	VAR robtarget OpenholeUD_3424 := [[417.35, -17.1, 182.09], [-0.110581, 0.698407, 0.70005, 0.099652], [0,0,0,0], [9E9, 9E9, 9E9, 9E9, 9E9, 9E9]];
	VAR robtarget OpenholeUD_3425 := [[421.34, -17.1, 182.02], [-0.098166, 0.70026, 0.701711, 0.087187], [0,0,0,0], [9E9, 9E9, 9E9, 9E9, 9E9, 9E9]];
	VAR robtarget OpenholeUD_3426 := [[425.34, -17.1, 181.95], [-0.085471, 0.701922, 0.703176, 0.074457], [0,0,0,0], [9E9, 9E9, 9E9, 9E9, 9E9, 9E9]];
	VAR robtarget OpenholeUD_3427 := [[429.34, -17.1, 181.87], [-0.072525, 0.703378, 0.704428, 0.061492], [0,0,0,0], [9E9, 9E9, 9E9, 9E9, 9E9, 9E9]];
	VAR robtarget OpenholeUD_3428 := [[433.34, -17.1, 181.8], [-0.059361, 0.704611, 0.705453, 0.048326], [0,0,0,0], [9E9, 9E9, 9E9, 9E9, 9E9, 9E9]];
	VAR robtarget OpenholeUD_3429 := [[437.34, -17.1, 181.72], [-0.046017, 0.705608, 0.70624, 0.034996], [0,0,0,0], [9E9, 9E9, 9E9, 9E9, 9E9, 9E9]];
	VAR robtarget OpenholeUD_3430 := [[443.05, -17.1, 181.62], [-0.02675, 0.706601, 0.706931, 0.015776], [0,0,0,0], [9E9, 9E9, 9E9, 9E9, 9E9, 9E9]];
	VAR robtarget OpenholeUD_3431 := [[443.05, -17.1, 181.62], [-0.02675, 0.706601, 0.706931, 0.015776], [0,0,0,0], [9E9, 9E9, 9E9, 9E9, 9E9, 9E9]];
	VAR robtarget OpenholeUD_3432 := [[443.48, -15.9, 181.68], [-0.029359, 0.706497, 0.707033, 0.010242], [0,0,0,0], [9E9, 9E9, 9E9, 9E9, 9E9, 9E9]];
	VAR robtarget OpenholeUD_3433 := [[439.48, -15.9, 181.8], [-0.042881, 0.705805, 0.706708, 0.023756], [0,0,0,0], [9E9, 9E9, 9E9, 9E9, 9E9, 9E9]];
	VAR robtarget OpenholeUD_3434 := [[435.48, -15.9, 181.92], [-0.056278, 0.704864, 0.706129, 0.037174], [0,0,0,0], [9E9, 9E9, 9E9, 9E9, 9E9, 9E9]];
	VAR robtarget OpenholeUD_3435 := [[431.49, -15.9, 182.04], [-0.06951, 0.703682, 0.705304, 0.050457], [0,0,0,0], [9E9, 9E9, 9E9, 9E9, 9E9, 9E9]];
	VAR robtarget OpenholeUD_3436 := [[427.49, -15.9, 182.16], [-0.082538, 0.702273, 0.704244, 0.063565], [0,0,0,0], [9E9, 9E9, 9E9, 9E9, 9E9, 9E9]];
	VAR robtarget OpenholeUD_3437 := [[423.49, -15.9, 182.28], [-0.095326, 0.700652, 0.702961, 0.076462], [0,0,0,0], [9E9, 9E9, 9E9, 9E9, 9E9, 9E9]];
	VAR robtarget OpenholeUD_3438 := [[419.49, -15.9, 182.4], [-0.107844, 0.698835, 0.701469, 0.089115], [0,0,0,0], [9E9, 9E9, 9E9, 9E9, 9E9, 9E9]];
	VAR robtarget OpenholeUD_3439 := [[415.49, -15.9, 182.52], [-0.120064, 0.696839, 0.699785, 0.101497], [0,0,0,0], [9E9, 9E9, 9E9, 9E9, 9E9, 9E9]];
	VAR robtarget OpenholeUD_3440 := [[411.5, -15.9, 182.64], [-0.131964, 0.694684, 0.697925, 0.113581], [0,0,0,0], [9E9, 9E9, 9E9, 9E9, 9E9, 9E9]];
	VAR robtarget OpenholeUD_3441 := [[407.5, -15.9, 182.76], [-0.143525, 0.692388, 0.695908, 0.125349], [0,0,0,0], [9E9, 9E9, 9E9, 9E9, 9E9, 9E9]];
	VAR robtarget OpenholeUD_3442 := [[403.5, -15.9, 182.88], [-0.154733, 0.689969, 0.693751, 0.136783], [0,0,0,0], [9E9, 9E9, 9E9, 9E9, 9E9, 9E9]];
	VAR robtarget OpenholeUD_3443 := [[399.5, -15.9, 183], [-0.165579, 0.687447, 0.691472, 0.147872], [0,0,0,0], [9E9, 9E9, 9E9, 9E9, 9E9, 9E9]];
	VAR robtarget OpenholeUD_3444 := [[395.5, -15.9, 183.12], [-0.176055, 0.684839, 0.689089, 0.158607], [0,0,0,0], [9E9, 9E9, 9E9, 9E9, 9E9, 9E9]];
	VAR robtarget OpenholeUD_3445 := [[389.35, -15.9, 183.31], [-0.191445, 0.680697, 0.685258, 0.174418], [0,0,0,0], [9E9, 9E9, 9E9, 9E9, 9E9, 9E9]];
	VAR robtarget OpenholeUD_3446 := [[385.35, -15.9, 183.32], [-0.183051, 0.683002, 0.683002, 0.183051], [0,0,0,0], [9E9, 9E9, 9E9, 9E9, 9E9, 9E9]];
	VAR robtarget OpenholeUD_3447 := [[381.35, -15.9, 183.33], [-0.183051, 0.683002, 0.683002, 0.183051], [0,0,0,0], [9E9, 9E9, 9E9, 9E9, 9E9, 9E9]];
	VAR robtarget OpenholeUD_3448 := [[377.35, -15.9, 183.34], [-0.183051, 0.683002, 0.683002, 0.183051], [0,0,0,0], [9E9, 9E9, 9E9, 9E9, 9E9, 9E9]];
	VAR robtarget OpenholeUD_3449 := [[369.35, -15.9, 183.37], [-0.183051, 0.683002, 0.683002, 0.183051], [0,0,0,0], [9E9, 9E9, 9E9, 9E9, 9E9, 9E9]];
	VAR robtarget OpenholeUD_3450 := [[369.35, -15.9, 183.37], [-0.183051, 0.683002, 0.683002, 0.183051], [0,0,0,0], [9E9, 9E9, 9E9, 9E9, 9E9, 9E9]];
	VAR robtarget OpenholeUD_3451 := [[369.35, -14.7, 184.06], [-0.183051, 0.683002, 0.683002, 0.183051], [0,0,0,0], [9E9, 9E9, 9E9, 9E9, 9E9, 9E9]];
	VAR robtarget OpenholeUD_3452 := [[373.35, -14.7, 184.05], [-0.183051, 0.683002, 0.683002, 0.183051], [0,0,0,0], [9E9, 9E9, 9E9, 9E9, 9E9, 9E9]];
	VAR robtarget OpenholeUD_3453 := [[377.35, -14.7, 184.04], [-0.183051, 0.683002, 0.683002, 0.183051], [0,0,0,0], [9E9, 9E9, 9E9, 9E9, 9E9, 9E9]];
	VAR robtarget OpenholeUD_3454 := [[381.35, -14.7, 184.03], [-0.183051, 0.683002, 0.683002, 0.183051], [0,0,0,0], [9E9, 9E9, 9E9, 9E9, 9E9, 9E9]];
	VAR robtarget OpenholeUD_3455 := [[389.35, -14.7, 184], [-0.194849, 0.679731, 0.68612, 0.170995], [0,0,0,0], [9E9, 9E9, 9E9, 9E9, 9E9, 9E9]];
	VAR robtarget OpenholeUD_3456 := [[393.35, -14.7, 183.83], [-0.185019, 0.682472, 0.688592, 0.16075], [0,0,0,0], [9E9, 9E9, 9E9, 9E9, 9E9, 9E9]];
	VAR robtarget OpenholeUD_3457 := [[397.35, -14.7, 183.67], [-0.174817, 0.685156, 0.690982, 0.150146], [0,0,0,0], [9E9, 9E9, 9E9, 9E9, 9E9, 9E9]];
	VAR robtarget OpenholeUD_3458 := [[401.34, -14.7, 183.5], [-0.164241, 0.687768, 0.693273, 0.139186], [0,0,0,0], [9E9, 9E9, 9E9, 9E9, 9E9, 9E9]];
	VAR robtarget OpenholeUD_3459 := [[405.34, -14.7, 183.33], [-0.153297, 0.69029, 0.695448, 0.127878], [0,0,0,0], [9E9, 9E9, 9E9, 9E9, 9E9, 9E9]];
	VAR robtarget OpenholeUD_3460 := [[409.34, -14.7, 183.17], [-0.141992, 0.692704, 0.697488, 0.116232], [0,0,0,0], [9E9, 9E9, 9E9, 9E9, 9E9, 9E9]];
	VAR robtarget OpenholeUD_3461 := [[413.33, -14.7, 183], [-0.130337, 0.694991, 0.699378, 0.104265], [0,0,0,0], [9E9, 9E9, 9E9, 9E9, 9E9, 9E9]];
	VAR robtarget OpenholeUD_3462 := [[417.33, -14.7, 182.83], [-0.118347, 0.697133, 0.701097, 0.091993], [0,0,0,0], [9E9, 9E9, 9E9, 9E9, 9E9, 9E9]];
	VAR robtarget OpenholeUD_3463 := [[421.33, -14.7, 182.67], [-0.106043, 0.69911, 0.70263, 0.07944], [0,0,0,0], [9E9, 9E9, 9E9, 9E9, 9E9, 9E9]];
	VAR robtarget OpenholeUD_3464 := [[425.32, -14.7, 182.5], [-0.093448, 0.700905, 0.70396, 0.066634], [0,0,0,0], [9E9, 9E9, 9E9, 9E9, 9E9, 9E9]];
	VAR robtarget OpenholeUD_3465 := [[429.32, -14.7, 182.34], [-0.080591, 0.702499, 0.705072, 0.053604], [0,0,0,0], [9E9, 9E9, 9E9, 9E9, 9E9, 9E9]];
	VAR robtarget OpenholeUD_3466 := [[433.32, -14.7, 182.17], [-0.067504, 0.703877, 0.705953, 0.040385], [0,0,0,0], [9E9, 9E9, 9E9, 9E9, 9E9, 9E9]];
	VAR robtarget OpenholeUD_3467 := [[437.31, -14.7, 182], [-0.054224, 0.705025, 0.706591, 0.027016], [0,0,0,0], [9E9, 9E9, 9E9, 9E9, 9E9, 9E9]];
	VAR robtarget OpenholeUD_3468 := [[444.22, -14.7, 181.71], [-0.030919, 0.70643, 0.707097, 0.003662], [0,0,0,0], [9E9, 9E9, 9E9, 9E9, 9E9, 9E9]];
	VAR robtarget OpenholeUD_3469 := [[444.22, -14.7, 181.71], [-0.030919, 0.70643, 0.707097, 0.003662], [0,0,0,0], [9E9, 9E9, 9E9, 9E9, 9E9, 9E9]];
	VAR robtarget OpenholeUD_3470 := [[445.45, -13.5, 181.71], [-0.030843, 0.706434, 0.707092, -0.004551], [0,0,0,0], [9E9, 9E9, 9E9, 9E9, 9E9, 9E9]];
	VAR robtarget OpenholeUD_3471 := [[441.45, -13.5, 181.92], [-0.044373, 0.705713, 0.70705, 0.009], [0,0,0,0], [9E9, 9E9, 9E9, 9E9, 9E9, 9E9]];
	VAR robtarget OpenholeUD_3472 := [[437.46, -13.5, 182.13], [-0.057785, 0.704742, 0.706749, 0.022491], [0,0,0,0], [9E9, 9E9, 9E9, 9E9, 9E9, 9E9]];
	VAR robtarget OpenholeUD_3473 := [[433.46, -13.5, 182.35], [-0.071038, 0.703529, 0.706196, 0.035882], [0,0,0,0], [9E9, 9E9, 9E9, 9E9, 9E9, 9E9]];
	VAR robtarget OpenholeUD_3474 := [[429.47, -13.5, 182.56], [-0.084092, 0.702089, 0.705398, 0.04913], [0,0,0,0], [9E9, 9E9, 9E9, 9E9, 9E9, 9E9]];
	VAR robtarget OpenholeUD_3475 := [[425.48, -13.5, 182.77], [-0.096912, 0.700434, 0.704366, 0.062197], [0,0,0,0], [9E9, 9E9, 9E9, 9E9, 9E9, 9E9]];
	VAR robtarget OpenholeUD_3476 := [[421.48, -13.5, 182.98], [-0.109465, 0.698582, 0.703113, 0.075049], [0,0,0,0], [9E9, 9E9, 9E9, 9E9, 9E9, 9E9]];
	VAR robtarget OpenholeUD_3477 := [[417.49, -13.5, 183.2], [-0.121724, 0.696551, 0.701653, 0.087653], [0,0,0,0], [9E9, 9E9, 9E9, 9E9, 9E9, 9E9]];
	VAR robtarget OpenholeUD_3478 := [[413.49, -13.5, 183.41], [-0.133665, 0.694358, 0.700003, 0.099981], [0,0,0,0], [9E9, 9E9, 9E9, 9E9, 9E9, 9E9]];
	VAR robtarget OpenholeUD_3479 := [[409.5, -13.5, 183.62], [-0.145268, 0.692024, 0.698179, 0.112012], [0,0,0,0], [9E9, 9E9, 9E9, 9E9, 9E9, 9E9]];
	VAR robtarget OpenholeUD_3480 := [[405.5, -13.5, 183.83], [-0.156519, 0.689566, 0.696199, 0.123724], [0,0,0,0], [9E9, 9E9, 9E9, 9E9, 9E9, 9E9]];
	VAR robtarget OpenholeUD_3481 := [[401.51, -13.5, 184.05], [-0.167407, 0.687004, 0.69408, 0.135103], [0,0,0,0], [9E9, 9E9, 9E9, 9E9, 9E9, 9E9]];
	VAR robtarget OpenholeUD_3482 := [[397.51, -13.5, 184.26], [-0.177925, 0.684356, 0.691841, 0.146136], [0,0,0,0], [9E9, 9E9, 9E9, 9E9, 9E9, 9E9]];
	VAR robtarget OpenholeUD_3483 := [[393.52, -13.5, 184.47], [-0.188069, 0.681638, 0.689499, 0.156817], [0,0,0,0], [9E9, 9E9, 9E9, 9E9, 9E9, 9E9]];
	VAR robtarget OpenholeUD_3484 := [[389.36, -13.5, 184.69], [-0.198245, 0.678748, 0.686964, 0.167571], [0,0,0,0], [9E9, 9E9, 9E9, 9E9, 9E9, 9E9]];
	VAR robtarget OpenholeUD_3485 := [[385.36, -13.5, 184.71], [-0.183051, 0.683002, 0.683002, 0.183051], [0,0,0,0], [9E9, 9E9, 9E9, 9E9, 9E9, 9E9]];
	VAR robtarget OpenholeUD_3486 := [[381.36, -13.5, 184.72], [-0.183051, 0.683002, 0.683002, 0.183051], [0,0,0,0], [9E9, 9E9, 9E9, 9E9, 9E9, 9E9]];
	VAR robtarget OpenholeUD_3487 := [[377.36, -13.5, 184.73], [-0.183051, 0.683002, 0.683002, 0.183051], [0,0,0,0], [9E9, 9E9, 9E9, 9E9, 9E9, 9E9]];
	VAR robtarget OpenholeUD_3488 := [[373.36, -13.5, 184.74], [-0.183051, 0.683002, 0.683002, 0.183051], [0,0,0,0], [9E9, 9E9, 9E9, 9E9, 9E9, 9E9]];
	VAR robtarget OpenholeUD_3489 := [[369.36, -13.5, 184.76], [-0.183051, 0.683002, 0.683002, 0.183051], [0,0,0,0], [9E9, 9E9, 9E9, 9E9, 9E9, 9E9]];
	VAR robtarget OpenholeUD_3490 := [[369.36, -13.5, 184.76], [-0.183051, 0.683002, 0.683002, 0.183051], [0,0,0,0], [9E9, 9E9, 9E9, 9E9, 9E9, 9E9]];
	VAR robtarget OpenholeUD_3491 := [[369.36, -12.3, 185.45], [-0.183051, 0.683002, 0.683002, 0.183051], [0,0,0,0], [9E9, 9E9, 9E9, 9E9, 9E9, 9E9]];
	VAR robtarget OpenholeUD_3492 := [[373.36, -12.3, 185.44], [-0.183051, 0.683002, 0.683002, 0.183051], [0,0,0,0], [9E9, 9E9, 9E9, 9E9, 9E9, 9E9]];
	VAR robtarget OpenholeUD_3493 := [[377.36, -12.3, 185.42], [-0.183051, 0.683002, 0.683002, 0.183051], [0,0,0,0], [9E9, 9E9, 9E9, 9E9, 9E9, 9E9]];
	VAR robtarget OpenholeUD_3494 := [[381.36, -12.3, 185.41], [-0.183051, 0.683002, 0.683002, 0.183051], [0,0,0,0], [9E9, 9E9, 9E9, 9E9, 9E9, 9E9]];
	VAR robtarget OpenholeUD_3495 := [[385.36, -12.3, 185.4], [-0.183051, 0.683002, 0.683002, 0.183051], [0,0,0,0], [9E9, 9E9, 9E9, 9E9, 9E9, 9E9]];
	VAR robtarget OpenholeUD_3496 := [[389.36, -12.3, 185.39], [-0.201634, 0.677749, 0.687791, 0.164145], [0,0,0,0], [9E9, 9E9, 9E9, 9E9, 9E9, 9E9]];
	VAR robtarget OpenholeUD_3497 := [[393.35, -12.3, 185.13], [-0.191956, 0.680553, 0.690183, 0.153776], [0,0,0,0], [9E9, 9E9, 9E9, 9E9, 9E9, 9E9]];
	VAR robtarget OpenholeUD_3498 := [[397.34, -12.3, 184.87], [-0.181904, 0.683309, 0.692486, 0.143051], [0,0,0,0], [9E9, 9E9, 9E9, 9E9, 9E9, 9E9]];
	VAR robtarget OpenholeUD_3499 := [[401.33, -12.3, 184.61], [-0.171477, 0.686, 0.694682, 0.131975], [0,0,0,0], [9E9, 9E9, 9E9, 9E9, 9E9, 9E9]];
	VAR robtarget OpenholeUD_3500 := [[405.33, -12.3, 184.35], [-0.160678, 0.688609, 0.696754, 0.120556], [0,0,0,0], [9E9, 9E9, 9E9, 9E9, 9E9, 9E9]];
	VAR robtarget OpenholeUD_3501 := [[409.32, -12.3, 184.09], [-0.149513, 0.691119, 0.698685, 0.108807], [0,0,0,0], [9E9, 9E9, 9E9, 9E9, 9E9, 9E9]];
	VAR robtarget OpenholeUD_3502 := [[413.31, -12.3, 183.84], [-0.137992, 0.693511, 0.700458, 0.096743], [0,0,0,0], [9E9, 9E9, 9E9, 9E9, 9E9, 9E9]];
	VAR robtarget OpenholeUD_3503 := [[417.3, -12.3, 183.58], [-0.12613, 0.695767, 0.702054, 0.084384], [0,0,0,0], [9E9, 9E9, 9E9, 9E9, 9E9, 9E9]];
	VAR robtarget OpenholeUD_3504 := [[421.29, -12.3, 183.32], [-0.113945, 0.697866, 0.703457, 0.071753], [0,0,0,0], [9E9, 9E9, 9E9, 9E9, 9E9, 9E9]];
	VAR robtarget OpenholeUD_3505 := [[425.28, -12.3, 183.06], [-0.10146, 0.69979, 0.704651, 0.058879], [0,0,0,0], [9E9, 9E9, 9E9, 9E9, 9E9, 9E9]];
	VAR robtarget OpenholeUD_3506 := [[429.28, -12.3, 182.8], [-0.088701, 0.701521, 0.705622, 0.045794], [0,0,0,0], [9E9, 9E9, 9E9, 9E9, 9E9, 9E9]];
	VAR robtarget OpenholeUD_3507 := [[433.27, -12.3, 182.54], [-0.0757, 0.703043, 0.706358, 0.032532], [0,0,0,0], [9E9, 9E9, 9E9, 9E9, 9E9, 9E9]];
	VAR robtarget OpenholeUD_3508 := [[437.26, -12.3, 182.28], [-0.062492, 0.70434, 0.706848, 0.019133], [0,0,0,0], [9E9, 9E9, 9E9, 9E9, 9E9, 9E9]];
	VAR robtarget OpenholeUD_3509 := [[441.25, -12.3, 182.03], [-0.049116, 0.705399, 0.707084, 0.005638], [0,0,0,0], [9E9, 9E9, 9E9, 9E9, 9E9, 9E9]];
	VAR robtarget OpenholeUD_3510 := [[445.24, -12.3, 181.77], [-0.035614, 0.706209, 0.707063, -0.007911], [0,0,0,0], [9E9, 9E9, 9E9, 9E9, 9E9, 9E9]];
	VAR robtarget OpenholeUD_3511 := [[449.23, -12.3, 181.51], [-0.022029, 0.706764, 0.706781, -0.021469], [0,0,0,0], [9E9, 9E9, 9E9, 9E9, 9E9, 9E9]];
	VAR robtarget OpenholeUD_3512 := [[453.22, -12.3, 181.25], [-0.008405, 0.707057, 0.706241, -0.034991], [0,0,0,0], [9E9, 9E9, 9E9, 9E9, 9E9, 9E9]];
	VAR robtarget OpenholeUD_3513 := [[457.22, -12.3, 180.99], [0.00521, 0.707088, 0.705446, -0.048433], [0,0,0,0], [9E9, 9E9, 9E9, 9E9, 9E9, 9E9]];
	VAR robtarget OpenholeUD_3514 := [[461.21, -12.3, 180.73], [0.018773, 0.706858, 0.704405, -0.061753], [0,0,0,0], [9E9, 9E9, 9E9, 9E9, 9E9, 9E9]];
	VAR robtarget OpenholeUD_3515 := [[465.2, -12.3, 180.47], [0.032238, 0.706372, 0.703128, -0.074909], [0,0,0,0], [9E9, 9E9, 9E9, 9E9, 9E9, 9E9]];
	VAR robtarget OpenholeUD_3516 := [[469.19, -12.3, 180.22], [0.045564, 0.705637, 0.701627, -0.087863], [0,0,0,0], [9E9, 9E9, 9E9, 9E9, 9E9, 9E9]];
	VAR robtarget OpenholeUD_3517 := [[473.18, -12.3, 179.96], [0.058713, 0.704665, 0.699917, -0.100581], [0,0,0,0], [9E9, 9E9, 9E9, 9E9, 9E9, 9E9]];
	VAR robtarget OpenholeUD_3518 := [[477.17, -12.3, 179.7], [0.071646, 0.703468, 0.698014, -0.113032], [0,0,0,0], [9E9, 9E9, 9E9, 9E9, 9E9, 9E9]];
	VAR robtarget OpenholeUD_3519 := [[481.17, -12.3, 179.44], [0.084333, 0.70206, 0.695937, -0.125188], [0,0,0,0], [9E9, 9E9, 9E9, 9E9, 9E9, 9E9]];
	VAR robtarget OpenholeUD_3520 := [[485.16, -12.3, 179.18], [0.096745, 0.700457, 0.693703, -0.137027], [0,0,0,0], [9E9, 9E9, 9E9, 9E9, 9E9, 9E9]];
	VAR robtarget OpenholeUD_3521 := [[489.15, -12.3, 178.92], [0.108857, 0.698677, 0.691331, -0.14853], [0,0,0,0], [9E9, 9E9, 9E9, 9E9, 9E9, 9E9]];
	VAR robtarget OpenholeUD_3522 := [[493.14, -12.3, 178.67], [0.12065, 0.696738, 0.68884, -0.159683], [0,0,0,0], [9E9, 9E9, 9E9, 9E9, 9E9, 9E9]];
	VAR robtarget OpenholeUD_3523 := [[497.13, -12.3, 178.41], [0.132108, 0.694656, 0.686249, -0.170476], [0,0,0,0], [9E9, 9E9, 9E9, 9E9, 9E9, 9E9]];
	VAR robtarget OpenholeUD_3524 := [[501.12, -12.3, 178.15], [0.143219, 0.692451, 0.683575, -0.180902], [0,0,0,0], [9E9, 9E9, 9E9, 9E9, 9E9, 9E9]];
	VAR robtarget OpenholeUD_3525 := [[505.12, -12.3, 177.89], [0.153974, 0.690139, 0.680835, -0.190956], [0,0,0,0], [9E9, 9E9, 9E9, 9E9, 9E9, 9E9]];
	VAR robtarget OpenholeUD_3526 := [[509.33, -12.3, 177.62], [0.183051, 0.683002, 0.683002, -0.183051], [0,0,0,0], [9E9, 9E9, 9E9, 9E9, 9E9, 9E9]];
	VAR robtarget OpenholeUD_3527 := [[513.33, -12.3, 177.6], [0.183051, 0.683002, 0.683002, -0.183051], [0,0,0,0], [9E9, 9E9, 9E9, 9E9, 9E9, 9E9]];
	VAR robtarget OpenholeUD_3528 := [[517.33, -12.3, 177.59], [0.183051, 0.683002, 0.683002, -0.183051], [0,0,0,0], [9E9, 9E9, 9E9, 9E9, 9E9, 9E9]];
	VAR robtarget OpenholeUD_3529 := [[521.33, -12.3, 177.58], [0.183051, 0.683002, 0.683002, -0.183051], [0,0,0,0], [9E9, 9E9, 9E9, 9E9, 9E9, 9E9]];
	VAR robtarget OpenholeUD_3530 := [[529.33, -12.3, 177.55], [0.183051, 0.683002, 0.683002, -0.183051], [0,0,0,0], [9E9, 9E9, 9E9, 9E9, 9E9, 9E9]];
	VAR robtarget OpenholeUD_3531 := [[529.33, -12.3, 177.55], [0.183051, 0.683002, 0.683002, -0.183051], [0,0,0,0], [9E9, 9E9, 9E9, 9E9, 9E9, 9E9]];
	VAR robtarget OpenholeUD_3532 := [[529.34, -13.5, 178.25], [0.183051, 0.683002, 0.683002, -0.183051], [0,0,0,0], [9E9, 9E9, 9E9, 9E9, 9E9, 9E9]];
	VAR robtarget OpenholeUD_3533 := [[525.34, -13.5, 178.26], [0.183051, 0.683002, 0.683002, -0.183051], [0,0,0,0], [9E9, 9E9, 9E9, 9E9, 9E9, 9E9]];
	VAR robtarget OpenholeUD_3534 := [[521.34, -13.5, 178.27], [0.183051, 0.683002, 0.683002, -0.183051], [0,0,0,0], [9E9, 9E9, 9E9, 9E9, 9E9, 9E9]];
	VAR robtarget OpenholeUD_3535 := [[517.34, -13.5, 178.28], [0.183051, 0.683002, 0.683002, -0.183051], [0,0,0,0], [9E9, 9E9, 9E9, 9E9, 9E9, 9E9]];
	VAR robtarget OpenholeUD_3536 := [[513.34, -13.5, 178.3], [0.183051, 0.683002, 0.683002, -0.183051], [0,0,0,0], [9E9, 9E9, 9E9, 9E9, 9E9, 9E9]];
	VAR robtarget OpenholeUD_3537 := [[509.34, -13.5, 178.31], [0.183051, 0.683002, 0.683002, -0.183051], [0,0,0,0], [9E9, 9E9, 9E9, 9E9, 9E9, 9E9]];
	VAR robtarget OpenholeUD_3538 := [[505.34, -13.5, 178.52], [0.158072, 0.689212, 0.681639, -0.188064], [0,0,0,0], [9E9, 9E9, 9E9, 9E9, 9E9, 9E9]];
	VAR robtarget OpenholeUD_3539 := [[501.35, -13.5, 178.73], [0.147397, 0.691574, 0.684348, -0.177955], [0,0,0,0], [9E9, 9E9, 9E9, 9E9, 9E9, 9E9]];
	VAR robtarget OpenholeUD_3540 := [[497.35, -13.5, 178.95], [0.136364, 0.693833, 0.686987, -0.167476], [0,0,0,0], [9E9, 9E9, 9E9, 9E9, 9E9, 9E9]];
	VAR robtarget OpenholeUD_3541 := [[493.36, -13.5, 179.16], [0.124981, 0.695974, 0.689541, -0.156632], [0,0,0,0], [9E9, 9E9, 9E9, 9E9, 9E9, 9E9]];
	VAR robtarget OpenholeUD_3542 := [[489.37, -13.5, 179.37], [0.113258, 0.697977, 0.69199, -0.145429], [0,0,0,0], [9E9, 9E9, 9E9, 9E9, 9E9, 9E9]];
	VAR robtarget OpenholeUD_3543 := [[485.37, -13.5, 179.58], [0.101212, 0.699826, 0.694317, -0.133878], [0,0,0,0], [9E9, 9E9, 9E9, 9E9, 9E9, 9E9]];
	VAR robtarget OpenholeUD_3544 := [[481.38, -13.5, 179.8], [0.08886, 0.701501, 0.696504, -0.121994], [0,0,0,0], [9E9, 9E9, 9E9, 9E9, 9E9, 9E9]];
	VAR robtarget OpenholeUD_3545 := [[477.38, -13.5, 180.01], [0.076227, 0.702986, 0.698531, -0.109795], [0,0,0,0], [9E9, 9E9, 9E9, 9E9, 9E9, 9E9]];
	VAR robtarget OpenholeUD_3546 := [[473.39, -13.5, 180.22], [0.063339, 0.704264, 0.70038, -0.097306], [0,0,0,0], [9E9, 9E9, 9E9, 9E9, 9E9, 9E9]];
	VAR robtarget OpenholeUD_3547 := [[469.39, -13.5, 180.43], [0.05023, 0.70532, 0.702033, -0.084552], [0,0,0,0], [9E9, 9E9, 9E9, 9E9, 9E9, 9E9]];
	VAR robtarget OpenholeUD_3548 := [[465.4, -13.5, 180.65], [0.036933, 0.706142, 0.703476, -0.071567], [0,0,0,0], [9E9, 9E9, 9E9, 9E9, 9E9, 9E9]];
	VAR robtarget OpenholeUD_3549 := [[461.4, -13.5, 180.86], [0.023489, 0.706717, 0.704692, -0.058384], [0,0,0,0], [9E9, 9E9, 9E9, 9E9, 9E9, 9E9]];
	VAR robtarget OpenholeUD_3550 := [[457.41, -13.5, 181.07], [0.009938, 0.707037, 0.705671, -0.045043], [0,0,0,0], [9E9, 9E9, 9E9, 9E9, 9E9, 9E9]];
	VAR robtarget OpenholeUD_3551 := [[453.25, -13.5, 181.29], [-0.004254, 0.707094, 0.706426, -0.03101], [0,0,0,0], [9E9, 9E9, 9E9, 9E9, 9E9, 9E9]];
	VAR robtarget OpenholeUD_3552 := [[453.25, -13.5, 181.29], [-0.004254, 0.707094, 0.706426, -0.03101], [0,0,0,0], [9E9, 9E9, 9E9, 9E9, 9E9, 9E9]];
	VAR robtarget OpenholeUD_3553 := [[454.47, -14.7, 181.29], [0.003998, 0.707095, 0.706423, -0.031085], [0,0,0,0], [9E9, 9E9, 9E9, 9E9, 9E9, 9E9]];
	VAR robtarget OpenholeUD_3554 := [[458.47, -14.7, 181.12], [0.017595, 0.706888, 0.705703, -0.04454], [0,0,0,0], [9E9, 9E9, 9E9, 9E9, 9E9, 9E9]];
	VAR robtarget OpenholeUD_3555 := [[462.46, -14.7, 180.96], [0.03111, 0.706422, 0.704735, -0.057872], [0,0,0,0], [9E9, 9E9, 9E9, 9E9, 9E9, 9E9]];
	VAR robtarget OpenholeUD_3556 := [[466.46, -14.7, 180.79], [0.0445, 0.705705, 0.703529, -0.071042], [0,0,0,0], [9E9, 9E9, 9E9, 9E9, 9E9, 9E9]];
	VAR robtarget OpenholeUD_3557 := [[470.46, -14.7, 180.62], [0.057724, 0.704747, 0.702098, -0.084011], [0,0,0,0], [9E9, 9E9, 9E9, 9E9, 9E9, 9E9]];
	VAR robtarget OpenholeUD_3558 := [[474.45, -14.7, 180.46], [0.070746, 0.703559, 0.700457, -0.096744], [0,0,0,0], [9E9, 9E9, 9E9, 9E9, 9E9, 9E9]];
	VAR robtarget OpenholeUD_3559 := [[478.45, -14.7, 180.29], [0.08353, 0.702156, 0.698622, -0.109212], [0,0,0,0], [9E9, 9E9, 9E9, 9E9, 9E9, 9E9]];
	VAR robtarget OpenholeUD_3560 := [[482.45, -14.7, 180.12], [0.096047, 0.700553, 0.69661, -0.121386], [0,0,0,0], [9E9, 9E9, 9E9, 9E9, 9E9, 9E9]];
	VAR robtarget OpenholeUD_3561 := [[486.44, -14.7, 179.96], [0.108271, 0.698768, 0.694439, -0.133245], [0,0,0,0], [9E9, 9E9, 9E9, 9E9, 9E9, 9E9]];
	VAR robtarget OpenholeUD_3562 := [[490.44, -14.7, 179.79], [0.120181, 0.696819, 0.692128, -0.14477], [0,0,0,0], [9E9, 9E9, 9E9, 9E9, 9E9, 9E9]];
	VAR robtarget OpenholeUD_3563 := [[494.44, -14.7, 179.62], [0.131758, 0.694723, 0.689696, -0.155946], [0,0,0,0], [9E9, 9E9, 9E9, 9E9, 9E9, 9E9]];
	VAR robtarget OpenholeUD_3564 := [[498.43, -14.7, 179.46], [0.142989, 0.692498, 0.687161, -0.166763], [0,0,0,0], [9E9, 9E9, 9E9, 9E9, 9E9, 9E9]];
	VAR robtarget OpenholeUD_3565 := [[502.43, -14.7, 179.29], [0.153865, 0.690163, 0.68454, -0.177214], [0,0,0,0], [9E9, 9E9, 9E9, 9E9, 9E9, 9E9]];
	VAR robtarget OpenholeUD_3566 := [[509.34, -14.7, 179], [0.183051, 0.683002, 0.683002, -0.183051], [0,0,0,0], [9E9, 9E9, 9E9, 9E9, 9E9, 9E9]];
	VAR robtarget OpenholeUD_3567 := [[513.34, -14.7, 178.99], [0.183051, 0.683002, 0.683002, -0.183051], [0,0,0,0], [9E9, 9E9, 9E9, 9E9, 9E9, 9E9]];
	VAR robtarget OpenholeUD_3568 := [[517.34, -14.7, 178.98], [0.183051, 0.683002, 0.683002, -0.183051], [0,0,0,0], [9E9, 9E9, 9E9, 9E9, 9E9, 9E9]];
	VAR robtarget OpenholeUD_3569 := [[521.34, -14.7, 178.97], [0.183051, 0.683002, 0.683002, -0.183051], [0,0,0,0], [9E9, 9E9, 9E9, 9E9, 9E9, 9E9]];
	VAR robtarget OpenholeUD_3570 := [[525.34, -14.7, 178.95], [0.183051, 0.683002, 0.683002, -0.183051], [0,0,0,0], [9E9, 9E9, 9E9, 9E9, 9E9, 9E9]];
	VAR robtarget OpenholeUD_3571 := [[529.34, -14.7, 178.94], [0.183051, 0.683002, 0.683002, -0.183051], [0,0,0,0], [9E9, 9E9, 9E9, 9E9, 9E9, 9E9]];
	VAR robtarget OpenholeUD_3572 := [[529.34, -14.7, 178.94], [0.183051, 0.683002, 0.683002, -0.183051], [0,0,0,0], [9E9, 9E9, 9E9, 9E9, 9E9, 9E9]];
	VAR robtarget OpenholeUD_3573 := [[529.34, -15.9, 179.63], [0.183051, 0.683002, 0.683002, -0.183051], [0,0,0,0], [9E9, 9E9, 9E9, 9E9, 9E9, 9E9]];
	VAR robtarget OpenholeUD_3574 := [[525.34, -15.9, 179.65], [0.183051, 0.683002, 0.683002, -0.183051], [0,0,0,0], [9E9, 9E9, 9E9, 9E9, 9E9, 9E9]];
	VAR robtarget OpenholeUD_3575 := [[521.34, -15.9, 179.66], [0.183051, 0.683002, 0.683002, -0.183051], [0,0,0,0], [9E9, 9E9, 9E9, 9E9, 9E9, 9E9]];
	VAR robtarget OpenholeUD_3576 := [[517.34, -15.9, 179.67], [0.183051, 0.683002, 0.683002, -0.183051], [0,0,0,0], [9E9, 9E9, 9E9, 9E9, 9E9, 9E9]];
	VAR robtarget OpenholeUD_3577 := [[513.34, -15.9, 179.68], [0.183051, 0.683002, 0.683002, -0.183051], [0,0,0,0], [9E9, 9E9, 9E9, 9E9, 9E9, 9E9]];
	VAR robtarget OpenholeUD_3578 := [[509.34, -15.9, 179.7], [0.183051, 0.683002, 0.683002, -0.183051], [0,0,0,0], [9E9, 9E9, 9E9, 9E9, 9E9, 9E9]];
	VAR robtarget OpenholeUD_3579 := [[505.34, -15.9, 179.82], [0.165066, 0.68757, 0.683512, -0.181139], [0,0,0,0], [9E9, 9E9, 9E9, 9E9, 9E9, 9E9]];
	VAR robtarget OpenholeUD_3580 := [[501.35, -15.9, 179.94], [0.154517, 0.690018, 0.686148, -0.170883], [0,0,0,0], [9E9, 9E9, 9E9, 9E9, 9E9, 9E9]];
	VAR robtarget OpenholeUD_3581 := [[497.35, -15.9, 180.06], [0.143606, 0.692371, 0.688706, -0.160261], [0,0,0,0], [9E9, 9E9, 9E9, 9E9, 9E9, 9E9]];
	VAR robtarget OpenholeUD_3582 := [[493.35, -15.9, 180.18], [0.132339, 0.694612, 0.69117, -0.149277], [0,0,0,0], [9E9, 9E9, 9E9, 9E9, 9E9, 9E9]];
	VAR robtarget OpenholeUD_3583 := [[489.35, -15.9, 180.3], [0.120727, 0.696725, 0.693522, -0.137938], [0,0,0,0], [9E9, 9E9, 9E9, 9E9, 9E9, 9E9]];
	VAR robtarget OpenholeUD_3584 := [[485.35, -15.9, 180.42], [0.108783, 0.698689, 0.695743, -0.126258], [0,0,0,0], [9E9, 9E9, 9E9, 9E9, 9E9, 9E9]];
	VAR robtarget OpenholeUD_3585 := [[481.35, -15.9, 180.54], [0.096525, 0.700488, 0.697815, -0.114252], [0,0,0,0], [9E9, 9E9, 9E9, 9E9, 9E9, 9E9]];
	VAR robtarget OpenholeUD_3586 := [[477.36, -15.9, 180.66], [0.083976, 0.702103, 0.69972, -0.10194], [0,0,0,0], [9E9, 9E9, 9E9, 9E9, 9E9, 9E9]];
	VAR robtarget OpenholeUD_3587 := [[473.36, -15.9, 180.78], [0.071163, 0.703517, 0.701439, -0.089347], [0,0,0,0], [9E9, 9E9, 9E9, 9E9, 9E9, 9E9]];
	VAR robtarget OpenholeUD_3588 := [[469.36, -15.9, 180.9], [0.058115, 0.704715, 0.702956, -0.076501], [0,0,0,0], [9E9, 9E9, 9E9, 9E9, 9E9, 9E9]];
	VAR robtarget OpenholeUD_3589 := [[465.36, -15.9, 181.02], [0.044867, 0.705682, 0.704256, -0.063435], [0,0,0,0], [9E9, 9E9, 9E9, 9E9, 9E9, 9E9]];
	VAR robtarget OpenholeUD_3590 := [[461.36, -15.9, 181.14], [0.031458, 0.706407, 0.705324, -0.050185], [0,0,0,0], [9E9, 9E9, 9E9, 9E9, 9E9, 9E9]];
	VAR robtarget OpenholeUD_3591 := [[455.21, -15.9, 181.32], [0.010611, 0.707027, 0.70649, -0.029534], [0,0,0,0], [9E9, 9E9, 9E9, 9E9, 9E9, 9E9]];
	VAR robtarget OpenholeUD_3592 := [[455.21, -15.9, 181.32], [0.010611, 0.707027, 0.70649, -0.029534], [0,0,0,0], [9E9, 9E9, 9E9, 9E9, 9E9, 9E9]];
	VAR robtarget OpenholeUD_3593 := [[455.65, -17.1, 181.38], [0.01617, 0.706922, 0.706593, -0.026938], [0,0,0,0], [9E9, 9E9, 9E9, 9E9, 9E9, 9E9]];
	VAR robtarget OpenholeUD_3594 := [[459.65, -17.1, 181.31], [0.029726, 0.706482, 0.705952, -0.040402], [0,0,0,0], [9E9, 9E9, 9E9, 9E9, 9E9, 9E9]];
	VAR robtarget OpenholeUD_3595 := [[463.65, -17.1, 181.24], [0.043173, 0.705788, 0.705061, -0.053745], [0,0,0,0], [9E9, 9E9, 9E9, 9E9, 9E9, 9E9]];
	VAR robtarget OpenholeUD_3596 := [[467.64, -17.1, 181.16], [0.056469, 0.704848, 0.703932, -0.066928], [0,0,0,0], [9E9, 9E9, 9E9, 9E9, 9E9, 9E9]];
	VAR robtarget OpenholeUD_3597 := [[471.64, -17.1, 181.09], [0.069574, 0.703676, 0.702577, -0.079912], [0,0,0,0], [9E9, 9E9, 9E9, 9E9, 9E9, 9E9]];
	VAR robtarget OpenholeUD_3598 := [[475.64, -17.1, 181.01], [0.082454, 0.702283, 0.701009, -0.092663], [0,0,0,0], [9E9, 9E9, 9E9, 9E9, 9E9, 9E9]];
	VAR robtarget OpenholeUD_3599 := [[479.64, -17.1, 180.94], [0.095076, 0.700686, 0.699245, -0.10515], [0,0,0,0], [9E9, 9E9, 9E9, 9E9, 9E9, 9E9]];
	VAR robtarget OpenholeUD_3600 := [[483.64, -17.1, 180.87], [0.107412, 0.698901, 0.697302, -0.117345], [0,0,0,0], [9E9, 9E9, 9E9, 9E9, 9E9, 9E9]];
	VAR robtarget OpenholeUD_3601 := [[487.64, -17.1, 180.79], [0.119439, 0.696946, 0.695198, -0.129227], [0,0,0,0], [9E9, 9E9, 9E9, 9E9, 9E9, 9E9]];
	VAR robtarget OpenholeUD_3602 := [[491.64, -17.1, 180.72], [0.131138, 0.69484, 0.692952, -0.140776], [0,0,0,0], [9E9, 9E9, 9E9, 9E9, 9E9, 9E9]];
	VAR robtarget OpenholeUD_3603 := [[495.64, -17.1, 180.64], [0.142494, 0.692601, 0.690581, -0.151979], [0,0,0,0], [9E9, 9E9, 9E9, 9E9, 9E9, 9E9]];
	VAR robtarget OpenholeUD_3604 := [[499.64, -17.1, 180.57], [0.153495, 0.690246, 0.688105, -0.162825], [0,0,0,0], [9E9, 9E9, 9E9, 9E9, 9E9, 9E9]];
	VAR robtarget OpenholeUD_3605 := [[503.64, -17.1, 180.49], [0.164134, 0.687794, 0.685539, -0.173308], [0,0,0,0], [9E9, 9E9, 9E9, 9E9, 9E9, 9E9]];
	VAR robtarget OpenholeUD_3606 := [[509.34, -17.1, 180.39], [0.183051, 0.683002, 0.683002, -0.183051], [0,0,0,0], [9E9, 9E9, 9E9, 9E9, 9E9, 9E9]];
	VAR robtarget OpenholeUD_3607 := [[513.34, -17.1, 180.38], [0.183051, 0.683002, 0.683002, -0.183051], [0,0,0,0], [9E9, 9E9, 9E9, 9E9, 9E9, 9E9]];
	VAR robtarget OpenholeUD_3608 := [[517.34, -17.1, 180.36], [0.183051, 0.683002, 0.683002, -0.183051], [0,0,0,0], [9E9, 9E9, 9E9, 9E9, 9E9, 9E9]];
	VAR robtarget OpenholeUD_3609 := [[521.34, -17.1, 180.35], [0.183051, 0.683002, 0.683002, -0.183051], [0,0,0,0], [9E9, 9E9, 9E9, 9E9, 9E9, 9E9]];
	VAR robtarget OpenholeUD_3610 := [[525.34, -17.1, 180.34], [0.183051, 0.683002, 0.683002, -0.183051], [0,0,0,0], [9E9, 9E9, 9E9, 9E9, 9E9, 9E9]];
	VAR robtarget OpenholeUD_3611 := [[529.34, -17.1, 180.33], [0.183051, 0.683002, 0.683002, -0.183051], [0,0,0,0], [9E9, 9E9, 9E9, 9E9, 9E9, 9E9]];
	VAR robtarget OpenholeUD_3612 := [[529.34, -17.1, 180.33], [0.183051, 0.683002, 0.683002, -0.183051], [0,0,0,0], [9E9, 9E9, 9E9, 9E9, 9E9, 9E9]];
	VAR robtarget OpenholeUD_3613 := [[529.35, -18.3, 181.02], [0.183051, 0.683002, 0.683002, -0.183051], [0,0,0,0], [9E9, 9E9, 9E9, 9E9, 9E9, 9E9]];
	VAR robtarget OpenholeUD_3614 := [[525.35, -18.3, 181.03], [0.183051, 0.683002, 0.683002, -0.183051], [0,0,0,0], [9E9, 9E9, 9E9, 9E9, 9E9, 9E9]];
	VAR robtarget OpenholeUD_3615 := [[521.35, -18.3, 181.04], [0.183051, 0.683002, 0.683002, -0.183051], [0,0,0,0], [9E9, 9E9, 9E9, 9E9, 9E9, 9E9]];
	VAR robtarget OpenholeUD_3616 := [[517.35, -18.3, 181.06], [0.183051, 0.683002, 0.683002, -0.183051], [0,0,0,0], [9E9, 9E9, 9E9, 9E9, 9E9, 9E9]];
	VAR robtarget OpenholeUD_3617 := [[513.35, -18.3, 181.07], [0.183051, 0.683002, 0.683002, -0.183051], [0,0,0,0], [9E9, 9E9, 9E9, 9E9, 9E9, 9E9]];
	VAR robtarget OpenholeUD_3618 := [[509.35, -18.3, 181.08], [0.183051, 0.683002, 0.683002, -0.183051], [0,0,0,0], [9E9, 9E9, 9E9, 9E9, 9E9, 9E9]];
	VAR robtarget OpenholeUD_3619 := [[505.35, -18.3, 181.11], [0.172055, 0.685855, 0.685315, -0.174194], [0,0,0,0], [9E9, 9E9, 9E9, 9E9, 9E9, 9E9]];
	VAR robtarget OpenholeUD_3620 := [[501.35, -18.3, 181.14], [0.161639, 0.688384, 0.687874, -0.163798], [0,0,0,0], [9E9, 9E9, 9E9, 9E9, 9E9, 9E9]];
	VAR robtarget OpenholeUD_3621 := [[497.35, -18.3, 181.17], [0.150857, 0.690827, 0.690347, -0.153038], [0,0,0,0], [9E9, 9E9, 9E9, 9E9, 9E9, 9E9]];
	VAR robtarget OpenholeUD_3622 := [[493.35, -18.3, 181.19], [0.139715, 0.693167, 0.692718, -0.141921], [0,0,0,0], [9E9, 9E9, 9E9, 9E9, 9E9, 9E9]];
	VAR robtarget OpenholeUD_3623 := [[489.35, -18.3, 181.22], [0.128221, 0.695384, 0.694969, -0.130454], [0,0,0,0], [9E9, 9E9, 9E9, 9E9, 9E9, 9E9]];
	VAR robtarget OpenholeUD_3624 := [[485.35, -18.3, 181.25], [0.116388, 0.697462, 0.697081, -0.118653], [0,0,0,0], [9E9, 9E9, 9E9, 9E9, 9E9, 9E9]];
	VAR robtarget OpenholeUD_3625 := [[481.35, -18.3, 181.28], [0.104234, 0.699382, 0.699036, -0.106533], [0,0,0,0], [9E9, 9E9, 9E9, 9E9, 9E9, 9E9]];
	VAR robtarget OpenholeUD_3626 := [[477.35, -18.3, 181.31], [0.091779, 0.701125, 0.700815, -0.094116], [0,0,0,0], [9E9, 9E9, 9E9, 9E9, 9E9, 9E9]];
	VAR robtarget OpenholeUD_3627 := [[473.35, -18.3, 181.33], [0.079048, 0.702674, 0.702403, -0.081429], [0,0,0,0], [9E9, 9E9, 9E9, 9E9, 9E9, 9E9]];
	VAR robtarget OpenholeUD_3628 := [[469.35, -18.3, 181.36], [0.066072, 0.704013, 0.703781, -0.068499], [0,0,0,0], [9E9, 9E9, 9E9, 9E9, 9E9, 9E9]];
	VAR robtarget OpenholeUD_3629 := [[465.35, -18.3, 181.39], [0.052884, 0.705126, 0.704936, -0.055363], [0,0,0,0], [9E9, 9E9, 9E9, 9E9, 9E9, 9E9]];
	VAR robtarget OpenholeUD_3630 := [[461.35, -18.3, 181.42], [0.03952, 0.706002, 0.705855, -0.042055], [0,0,0,0], [9E9, 9E9, 9E9, 9E9, 9E9, 9E9]];
	VAR robtarget OpenholeUD_3631 := [[455.83, -18.3, 181.46], [0.020892, 0.706798, 0.706716, -0.023509], [0,0,0,0], [9E9, 9E9, 9E9, 9E9, 9E9, 9E9]];
	VAR robtarget OpenholeUD_3632 := [[455.83, -18.3, 181.46], [0.020892, 0.706798, 0.706716, -0.023509], [0,0,0,0], [9E9, 9E9, 9E9, 9E9, 9E9, 9E9]];
	VAR robtarget OpenholeUD_3633 := [[455.8, -19.5, 181.53], [0.024849, 0.70667, 0.706843, -0.01932], [0,0,0,0], [9E9, 9E9, 9E9, 9E9, 9E9, 9E9]];
	VAR robtarget OpenholeUD_3634 := [[459.8, -19.5, 181.55], [0.038371, 0.706065, 0.706345, -0.032813], [0,0,0,0], [9E9, 9E9, 9E9, 9E9, 9E9, 9E9]];
	VAR robtarget OpenholeUD_3635 := [[463.8, -19.5, 181.57], [0.051768, 0.705209, 0.705596, -0.046199], [0,0,0,0], [9E9, 9E9, 9E9, 9E9, 9E9, 9E9]];
	VAR robtarget OpenholeUD_3636 := [[467.8, -19.5, 181.59], [0.064998, 0.704113, 0.704604, -0.059436], [0,0,0,0], [9E9, 9E9, 9E9, 9E9, 9E9, 9E9]];
	VAR robtarget OpenholeUD_3637 := [[471.8, -19.5, 181.6], [0.078024, 0.702789, 0.703382, -0.072486], [0,0,0,0], [9E9, 9E9, 9E9, 9E9, 9E9, 9E9]];
	VAR robtarget OpenholeUD_3638 := [[475.8, -19.5, 181.62], [0.09081, 0.701251, 0.701941, -0.085312], [0,0,0,0], [9E9, 9E9, 9E9, 9E9, 9E9, 9E9]];
	VAR robtarget OpenholeUD_3639 := [[479.8, -19.5, 181.64], [0.103327, 0.699517, 0.700299, -0.097884], [0,0,0,0], [9E9, 9E9, 9E9, 9E9, 9E9, 9E9]];
	VAR robtarget OpenholeUD_3640 := [[483.8, -19.5, 181.66], [0.115547, 0.697602, 0.698471, -0.110174], [0,0,0,0], [9E9, 9E9, 9E9, 9E9, 9E9, 9E9]];
	VAR robtarget OpenholeUD_3641 := [[487.8, -19.5, 181.68], [0.127449, 0.695526, 0.696475, -0.122157], [0,0,0,0], [9E9, 9E9, 9E9, 9E9, 9E9, 9E9]];
	VAR robtarget OpenholeUD_3642 := [[491.8, -19.5, 181.69], [0.139015, 0.693307, 0.694329, -0.133815], [0,0,0,0], [9E9, 9E9, 9E9, 9E9, 9E9, 9E9]];
	VAR robtarget OpenholeUD_3643 := [[495.8, -19.5, 181.71], [0.150231, 0.690964, 0.692052, -0.145133], [0,0,0,0], [9E9, 9E9, 9E9, 9E9, 9E9, 9E9]];
	VAR robtarget OpenholeUD_3644 := [[499.8, -19.5, 181.73], [0.161087, 0.688514, 0.689662, -0.156097], [0,0,0,0], [9E9, 9E9, 9E9, 9E9, 9E9, 9E9]];
	VAR robtarget OpenholeUD_3645 := [[503.8, -19.5, 181.75], [0.171576, 0.685975, 0.687176, -0.166702], [0,0,0,0], [9E9, 9E9, 9E9, 9E9, 9E9, 9E9]];
	VAR robtarget OpenholeUD_3646 := [[509.35, -19.5, 181.77], [0.183051, 0.683002, 0.683002, -0.183051], [0,0,0,0], [9E9, 9E9, 9E9, 9E9, 9E9, 9E9]];
	VAR robtarget OpenholeUD_3647 := [[513.35, -19.5, 181.76], [0.183051, 0.683002, 0.683002, -0.183051], [0,0,0,0], [9E9, 9E9, 9E9, 9E9, 9E9, 9E9]];
	VAR robtarget OpenholeUD_3648 := [[517.35, -19.5, 181.75], [0.183051, 0.683002, 0.683002, -0.183051], [0,0,0,0], [9E9, 9E9, 9E9, 9E9, 9E9, 9E9]];
	VAR robtarget OpenholeUD_3649 := [[521.35, -19.5, 181.74], [0.183051, 0.683002, 0.683002, -0.183051], [0,0,0,0], [9E9, 9E9, 9E9, 9E9, 9E9, 9E9]];
	VAR robtarget OpenholeUD_3650 := [[525.35, -19.5, 181.72], [0.183051, 0.683002, 0.683002, -0.183051], [0,0,0,0], [9E9, 9E9, 9E9, 9E9, 9E9, 9E9]];
	VAR robtarget OpenholeUD_3651 := [[529.35, -19.5, 181.71], [0.183051, 0.683002, 0.683002, -0.183051], [0,0,0,0], [9E9, 9E9, 9E9, 9E9, 9E9, 9E9]];
	VAR robtarget OpenholeUD_3652 := [[529.35, -19.5, 181.71], [0.183051, 0.683002, 0.683002, -0.183051], [0,0,0,0], [9E9, 9E9, 9E9, 9E9, 9E9, 9E9]];
	VAR robtarget OpenholeUD_3653 := [[529.35, -20.7, 182.41], [0.183051, 0.683002, 0.683002, -0.183051], [0,0,0,0], [9E9, 9E9, 9E9, 9E9, 9E9, 9E9]];
	VAR robtarget OpenholeUD_3654 := [[525.35, -20.7, 182.42], [0.183051, 0.683002, 0.683002, -0.183051], [0,0,0,0], [9E9, 9E9, 9E9, 9E9, 9E9, 9E9]];
	VAR robtarget OpenholeUD_3655 := [[521.35, -20.7, 182.43], [0.183051, 0.683002, 0.683002, -0.183051], [0,0,0,0], [9E9, 9E9, 9E9, 9E9, 9E9, 9E9]];
	VAR robtarget OpenholeUD_3656 := [[517.35, -20.7, 182.44], [0.183051, 0.683002, 0.683002, -0.183051], [0,0,0,0], [9E9, 9E9, 9E9, 9E9, 9E9, 9E9]];
	VAR robtarget OpenholeUD_3657 := [[509.35, -20.7, 182.47], [0.183051, 0.683002, 0.683002, -0.183051], [0,0,0,0], [9E9, 9E9, 9E9, 9E9, 9E9, 9E9]];
	VAR robtarget OpenholeUD_3658 := [[505.35, -20.7, 182.4], [0.179031, 0.684067, 0.687046, -0.167237], [0,0,0,0], [9E9, 9E9, 9E9, 9E9, 9E9, 9E9]];
	VAR robtarget OpenholeUD_3659 := [[501.35, -20.7, 182.34], [0.168754, 0.686675, 0.689524, -0.156706], [0,0,0,0], [9E9, 9E9, 9E9, 9E9, 9E9, 9E9]];
	VAR robtarget OpenholeUD_3660 := [[497.35, -20.7, 182.27], [0.158109, 0.689204, 0.691909, -0.145816], [0,0,0,0], [9E9, 9E9, 9E9, 9E9, 9E9, 9E9]];
	VAR robtarget OpenholeUD_3661 := [[493.35, -20.7, 182.21], [0.147099, 0.691637, 0.694183, -0.134572], [0,0,0,0], [9E9, 9E9, 9E9, 9E9, 9E9, 9E9]];
	VAR robtarget OpenholeUD_3662 := [[489.35, -20.7, 182.15], [0.135731, 0.693957, 0.696329, -0.122985], [0,0,0,0], [9E9, 9E9, 9E9, 9E9, 9E9, 9E9]];
	VAR robtarget OpenholeUD_3663 := [[485.35, -20.7, 182.08], [0.124019, 0.696146, 0.698329, -0.11107], [0,0,0,0], [9E9, 9E9, 9E9, 9E9, 9E9, 9E9]];
	VAR robtarget OpenholeUD_3664 := [[481.35, -20.7, 182.02], [0.111977, 0.698184, 0.700164, -0.098845], [0,0,0,0], [9E9, 9E9, 9E9, 9E9, 9E9, 9E9]];
	VAR robtarget OpenholeUD_3665 := [[477.35, -20.7, 181.95], [0.099625, 0.700054, 0.701817, -0.086333], [0,0,0,0], [9E9, 9E9, 9E9, 9E9, 9E9, 9E9]];
	VAR robtarget OpenholeUD_3666 := [[473.35, -20.7, 181.89], [0.086987, 0.701736, 0.70327, -0.07356], [0,0,0,0], [9E9, 9E9, 9E9, 9E9, 9E9, 9E9]];
	VAR robtarget OpenholeUD_3667 := [[469.36, -20.7, 181.82], [0.074092, 0.703214, 0.704509, -0.060557], [0,0,0,0], [9E9, 9E9, 9E9, 9E9, 9E9, 9E9]];
	VAR robtarget OpenholeUD_3668 := [[465.36, -20.7, 181.76], [0.060972, 0.704473, 0.705519, -0.047359], [0,0,0,0], [9E9, 9E9, 9E9, 9E9, 9E9, 9E9]];
	VAR robtarget OpenholeUD_3669 := [[461.36, -20.7, 181.69], [0.047664, 0.705499, 0.706289, -0.034003], [0,0,0,0], [9E9, 9E9, 9E9, 9E9, 9E9, 9E9]];
	VAR robtarget OpenholeUD_3670 := [[455.53, -20.7, 181.6], [0.02803, 0.706551, 0.706961, -0.014357], [0,0,0,0], [9E9, 9E9, 9E9, 9E9, 9E9, 9E9]];
	VAR robtarget OpenholeUD_3671 := [[455.53, -20.7, 181.6], [0.02803, 0.706551, 0.706961, -0.014357], [0,0,0,0], [9E9, 9E9, 9E9, 9E9, 9E9, 9E9]];
	VAR robtarget OpenholeUD_3672 := [[455.01, -21.9, 181.66], [0.030322, 0.706456, 0.707056, -0.008506], [0,0,0,0], [9E9, 9E9, 9E9, 9E9, 9E9, 9E9]];
	VAR robtarget OpenholeUD_3673 := [[459, -21.9, 181.77], [0.043828, 0.705747, 0.706763, -0.022037], [0,0,0,0], [9E9, 9E9, 9E9, 9E9, 9E9, 9E9]];
	VAR robtarget OpenholeUD_3674 := [[463, -21.9, 181.88], [0.057201, 0.704789, 0.706216, -0.035483], [0,0,0,0], [9E9, 9E9, 9E9, 9E9, 9E9, 9E9]];
	VAR robtarget OpenholeUD_3675 := [[467, -21.9, 181.99], [0.070403, 0.703593, 0.705421, -0.048803], [0,0,0,0], [9E9, 9E9, 9E9, 9E9, 9E9, 9E9]];
	VAR robtarget OpenholeUD_3676 := [[471, -21.9, 182.1], [0.083395, 0.702172, 0.704387, -0.061955], [0,0,0,0], [9E9, 9E9, 9E9, 9E9, 9E9, 9E9]];
	VAR robtarget OpenholeUD_3677 := [[475, -21.9, 182.21], [0.096142, 0.70054, 0.703128, -0.074904], [0,0,0,0], [9E9, 9E9, 9E9, 9E9, 9E9, 9E9]];
	VAR robtarget OpenholeUD_3678 := [[479, -21.9, 182.32], [0.108614, 0.698715, 0.701658, -0.087616], [0,0,0,0], [9E9, 9E9, 9E9, 9E9, 9E9, 9E9]];
	VAR robtarget OpenholeUD_3679 := [[482.99, -21.9, 182.43], [0.120786, 0.696714, 0.699991, -0.10006], [0,0,0,0], [9E9, 9E9, 9E9, 9E9, 9E9, 9E9]];
	VAR robtarget OpenholeUD_3680 := [[486.99, -21.9, 182.54], [0.132635, 0.694556, 0.698146, -0.112212], [0,0,0,0], [9E9, 9E9, 9E9, 9E9, 9E9, 9E9]];
	VAR robtarget OpenholeUD_3681 := [[490.99, -21.9, 182.65], [0.144144, 0.692259, 0.69614, -0.12405], [0,0,0,0], [9E9, 9E9, 9E9, 9E9, 9E9, 9E9]];
	VAR robtarget OpenholeUD_3682 := [[494.99, -21.9, 182.76], [0.1553, 0.689842, 0.693992, -0.135557], [0,0,0,0], [9E9, 9E9, 9E9, 9E9, 9E9, 9E9]];
	VAR robtarget OpenholeUD_3683 := [[498.99, -21.9, 182.87], [0.166092, 0.687323, 0.691718, -0.146719], [0,0,0,0], [9E9, 9E9, 9E9, 9E9, 9E9, 9E9]];
	VAR robtarget OpenholeUD_3684 := [[502.99, -21.9, 182.98], [0.176516, 0.68472, 0.689337, -0.157526], [0,0,0,0], [9E9, 9E9, 9E9, 9E9, 9E9, 9E9]];
	VAR robtarget OpenholeUD_3685 := [[509.35, -21.9, 183.16], [0.183051, 0.683002, 0.683002, -0.183051], [0,0,0,0], [9E9, 9E9, 9E9, 9E9, 9E9, 9E9]];
	VAR robtarget OpenholeUD_3686 := [[513.35, -21.9, 183.15], [0.183051, 0.683002, 0.683002, -0.183051], [0,0,0,0], [9E9, 9E9, 9E9, 9E9, 9E9, 9E9]];
	VAR robtarget OpenholeUD_3687 := [[517.35, -21.9, 183.14], [0.183051, 0.683002, 0.683002, -0.183051], [0,0,0,0], [9E9, 9E9, 9E9, 9E9, 9E9, 9E9]];
	VAR robtarget OpenholeUD_3688 := [[521.35, -21.9, 183.12], [0.183051, 0.683002, 0.683002, -0.183051], [0,0,0,0], [9E9, 9E9, 9E9, 9E9, 9E9, 9E9]];
	VAR robtarget OpenholeUD_3689 := [[529.35, -21.9, 183.1], [0.183051, 0.683002, 0.683002, -0.183051], [0,0,0,0], [9E9, 9E9, 9E9, 9E9, 9E9, 9E9]];
	VAR robtarget OpenholeUD_3690 := [[529.35, -21.9, 183.1], [0.183051, 0.683002, 0.683002, -0.183051], [0,0,0,0], [9E9, 9E9, 9E9, 9E9, 9E9, 9E9]];
	VAR robtarget OpenholeUD_3691 := [[529.35, -23.1, 183.79], [0.183051, 0.683002, 0.683002, -0.183051], [0,0,0,0], [9E9, 9E9, 9E9, 9E9, 9E9, 9E9]];
	VAR robtarget OpenholeUD_3692 := [[525.35, -23.1, 183.8], [0.183051, 0.683002, 0.683002, -0.183051], [0,0,0,0], [9E9, 9E9, 9E9, 9E9, 9E9, 9E9]];
	VAR robtarget OpenholeUD_3693 := [[521.35, -23.1, 183.82], [0.183051, 0.683002, 0.683002, -0.183051], [0,0,0,0], [9E9, 9E9, 9E9, 9E9, 9E9, 9E9]];
	VAR robtarget OpenholeUD_3694 := [[517.35, -23.1, 183.83], [0.183051, 0.683002, 0.683002, -0.183051], [0,0,0,0], [9E9, 9E9, 9E9, 9E9, 9E9, 9E9]];
	VAR robtarget OpenholeUD_3695 := [[513.35, -23.1, 183.84], [0.183051, 0.683002, 0.683002, -0.183051], [0,0,0,0], [9E9, 9E9, 9E9, 9E9, 9E9, 9E9]];
	VAR robtarget OpenholeUD_3696 := [[509.35, -23.1, 183.85], [0.183051, 0.683002, 0.683002, -0.183051], [0,0,0,0], [9E9, 9E9, 9E9, 9E9, 9E9, 9E9]];
	VAR robtarget OpenholeUD_3697 := [[505.36, -23.1, 183.7], [0.185988, 0.682208, 0.688704, -0.160273], [0,0,0,0], [9E9, 9E9, 9E9, 9E9, 9E9, 9E9]];
	VAR robtarget OpenholeUD_3698 := [[501.36, -23.1, 183.54], [0.175857, 0.68489, 0.691097, -0.149615], [0,0,0,0], [9E9, 9E9, 9E9, 9E9, 9E9, 9E9]];
	VAR robtarget OpenholeUD_3699 := [[497.36, -23.1, 183.38], [0.165354, 0.687501, 0.69339, -0.138601], [0,0,0,0], [9E9, 9E9, 9E9, 9E9, 9E9, 9E9]];
	VAR robtarget OpenholeUD_3700 := [[493.37, -23.1, 183.23], [0.154483, 0.690025, 0.695565, -0.127239], [0,0,0,0], [9E9, 9E9, 9E9, 9E9, 9E9, 9E9]];
	VAR robtarget OpenholeUD_3701 := [[489.37, -23.1, 183.07], [0.14325, 0.692445, 0.697603, -0.11554], [0,0,0,0], [9E9, 9E9, 9E9, 9E9, 9E9, 9E9]];
	VAR robtarget OpenholeUD_3702 := [[485.37, -23.1, 182.91], [0.131665, 0.69474, 0.699488, -0.103521], [0,0,0,0], [9E9, 9E9, 9E9, 9E9, 9E9, 9E9]];
	VAR robtarget OpenholeUD_3703 := [[481.38, -23.1, 182.76], [0.119743, 0.696894, 0.701201, -0.0912], [0,0,0,0], [9E9, 9E9, 9E9, 9E9, 9E9, 9E9]];
	VAR robtarget OpenholeUD_3704 := [[477.38, -23.1, 182.6], [0.107503, 0.698887, 0.702725, -0.078601], [0,0,0,0], [9E9, 9E9, 9E9, 9E9, 9E9, 9E9]];
	VAR robtarget OpenholeUD_3705 := [[473.38, -23.1, 182.44], [0.094967, 0.700701, 0.704043, -0.065752], [0,0,0,0], [9E9, 9E9, 9E9, 9E9, 9E9, 9E9]];
	VAR robtarget OpenholeUD_3706 := [[469.39, -23.1, 182.29], [0.082163, 0.702317, 0.705141, -0.052684], [0,0,0,0], [9E9, 9E9, 9E9, 9E9, 9E9, 9E9]];
	VAR robtarget OpenholeUD_3707 := [[465.39, -23.1, 182.13], [0.069122, 0.70372, 0.706006, -0.039434], [0,0,0,0], [9E9, 9E9, 9E9, 9E9, 9E9, 9E9]];
	VAR robtarget OpenholeUD_3708 := [[461.39, -23.1, 181.97], [0.055879, 0.704895, 0.706627, -0.02604], [0,0,0,0], [9E9, 9E9, 9E9, 9E9, 9E9, 9E9]];
	VAR robtarget OpenholeUD_3709 := [[454.13, -23.1, 181.69], [0.031439, 0.706408, 0.707105, -0.00148], [0,0,0,0], [9E9, 9E9, 9E9, 9E9, 9E9, 9E9]];
	VAR robtarget OpenholeUD_3710 := [[454.13, -23.1, 181.69], [0.031439, 0.706408, 0.707105, -0.00148], [0,0,0,0], [9E9, 9E9, 9E9, 9E9, 9E9, 9E9]];
	VAR robtarget OpenholeUD_3711 := [[452.65, -24.3, 181.67], [0.030476, 0.70645, 0.707066, 0.007623], [0,0,0,0], [9E9, 9E9, 9E9, 9E9, 9E9, 9E9]];
	VAR robtarget OpenholeUD_3712 := [[456.64, -24.3, 181.87], [0.044002, 0.705736, 0.707082, -0.005941], [0,0,0,0], [9E9, 9E9, 9E9, 9E9, 9E9, 9E9]];
	VAR robtarget OpenholeUD_3713 := [[460.64, -24.3, 182.07], [0.057407, 0.704773, 0.706839, -0.019461], [0,0,0,0], [9E9, 9E9, 9E9, 9E9, 9E9, 9E9]];
	VAR robtarget OpenholeUD_3714 := [[464.63, -24.3, 182.28], [0.070649, 0.703569, 0.706341, -0.032893], [0,0,0,0], [9E9, 9E9, 9E9, 9E9, 9E9, 9E9]];
	VAR robtarget OpenholeUD_3715 := [[468.63, -24.3, 182.48], [0.083691, 0.702137, 0.705596, -0.046195], [0,0,0,0], [9E9, 9E9, 9E9, 9E9, 9E9, 9E9]];
	VAR robtarget OpenholeUD_3716 := [[472.62, -24.3, 182.68], [0.096497, 0.700492, 0.704613, -0.059328], [0,0,0,0], [9E9, 9E9, 9E9, 9E9, 9E9, 9E9]];
	VAR robtarget OpenholeUD_3717 := [[476.62, -24.3, 182.89], [0.109034, 0.69865, 0.703405, -0.072256], [0,0,0,0], [9E9, 9E9, 9E9, 9E9, 9E9, 9E9]];
	VAR robtarget OpenholeUD_3718 := [[480.61, -24.3, 183.09], [0.121276, 0.696629, 0.701986, -0.084945], [0,0,0,0], [9E9, 9E9, 9E9, 9E9, 9E9, 9E9]];
	VAR robtarget OpenholeUD_3719 := [[484.61, -24.3, 183.29], [0.133199, 0.694448, 0.700371, -0.097366], [0,0,0,0], [9E9, 9E9, 9E9, 9E9, 9E9, 9E9]];
	VAR robtarget OpenholeUD_3720 := [[488.6, -24.3, 183.49], [0.144785, 0.692125, 0.698578, -0.109494], [0,0,0,0], [9E9, 9E9, 9E9, 9E9, 9E9, 9E9]];
	VAR robtarget OpenholeUD_3721 := [[492.6, -24.3, 183.7], [0.156019, 0.68968, 0.696623, -0.121309], [0,0,0,0], [9E9, 9E9, 9E9, 9E9, 9E9, 9E9]];
	VAR robtarget OpenholeUD_3722 := [[496.59, -24.3, 183.9], [0.16689, 0.68713, 0.694526, -0.132793], [0,0,0,0], [9E9, 9E9, 9E9, 9E9, 9E9, 9E9]];
	VAR robtarget OpenholeUD_3723 := [[500.59, -24.3, 184.1], [0.177392, 0.684494, 0.692303, -0.143935], [0,0,0,0], [9E9, 9E9, 9E9, 9E9, 9E9, 9E9]];
	VAR robtarget OpenholeUD_3724 := [[504.58, -24.3, 184.3], [0.187521, 0.681789, 0.689972, -0.154723], [0,0,0,0], [9E9, 9E9, 9E9, 9E9, 9E9, 9E9]];
	VAR robtarget OpenholeUD_3725 := [[509.36, -24.3, 184.55], [0.183051, 0.683002, 0.683002, -0.183051], [0,0,0,0], [9E9, 9E9, 9E9, 9E9, 9E9, 9E9]];
	VAR robtarget OpenholeUD_3726 := [[513.36, -24.3, 184.53], [0.183051, 0.683002, 0.683002, -0.183051], [0,0,0,0], [9E9, 9E9, 9E9, 9E9, 9E9, 9E9]];
	VAR robtarget OpenholeUD_3727 := [[517.36, -24.3, 184.52], [0.183051, 0.683002, 0.683002, -0.183051], [0,0,0,0], [9E9, 9E9, 9E9, 9E9, 9E9, 9E9]];
	VAR robtarget OpenholeUD_3728 := [[521.36, -24.3, 184.51], [0.183051, 0.683002, 0.683002, -0.183051], [0,0,0,0], [9E9, 9E9, 9E9, 9E9, 9E9, 9E9]];
	VAR robtarget OpenholeUD_3729 := [[525.36, -24.3, 184.5], [0.183051, 0.683002, 0.683002, -0.183051], [0,0,0,0], [9E9, 9E9, 9E9, 9E9, 9E9, 9E9]];
	VAR robtarget OpenholeUD_3730 := [[529.36, -24.3, 184.48], [0.183051, 0.683002, 0.683002, -0.183051], [0,0,0,0], [9E9, 9E9, 9E9, 9E9, 9E9, 9E9]];
	VAR robtarget OpenholeUD_3731 := [[529.35, -20.84, 182.48], [0.183051, 0.683002, 0.683002, -0.183051], [0,0,0,0], [9E9, 9E9, 9E9, 9E9, 9E9, 9E9]];
	VAR robtarget OpenholeUD_3732 := [[529.34, -17.37, 180.48], [0.183051, 0.683002, 0.683002, -0.183051], [0,0,0,0], [9E9, 9E9, 9E9, 9E9, 9E9, 9E9]];
	VAR robtarget OpenholeUD_3733 := [[529.33, -11.1, 176.86], [0.183051, 0.683002, 0.683002, -0.183051], [0,0,0,0], [9E9, 9E9, 9E9, 9E9, 9E9, 9E9]];
	VAR robtarget OpenholeUD_3734 := [[525.33, -11.1, 176.87], [0.183051, 0.683002, 0.683002, -0.183051], [0,0,0,0], [9E9, 9E9, 9E9, 9E9, 9E9, 9E9]];
	VAR robtarget OpenholeUD_3735 := [[521.33, -11.1, 176.89], [0.183051, 0.683002, 0.683002, -0.183051], [0,0,0,0], [9E9, 9E9, 9E9, 9E9, 9E9, 9E9]];
	VAR robtarget OpenholeUD_3736 := [[517.33, -11.1, 176.9], [0.183051, 0.683002, 0.683002, -0.183051], [0,0,0,0], [9E9, 9E9, 9E9, 9E9, 9E9, 9E9]];
	VAR robtarget OpenholeUD_3737 := [[513.33, -11.1, 176.91], [0.183051, 0.683002, 0.683002, -0.183051], [0,0,0,0], [9E9, 9E9, 9E9, 9E9, 9E9, 9E9]];
	VAR robtarget OpenholeUD_3738 := [[509.33, -11.1, 176.92], [0.183051, 0.683002, 0.683002, -0.183051], [0,0,0,0], [9E9, 9E9, 9E9, 9E9, 9E9, 9E9]];
	VAR robtarget OpenholeUD_3739 := [[505.34, -11.1, 177.23], [0.151079, 0.690779, 0.679698, -0.194963], [0,0,0,0], [9E9, 9E9, 9E9, 9E9, 9E9, 9E9]];
	VAR robtarget OpenholeUD_3740 := [[501.36, -11.1, 177.53], [0.140286, 0.693051, 0.682476, -0.185006], [0,0,0,0], [9E9, 9E9, 9E9, 9E9, 9E9, 9E9]];
	VAR robtarget OpenholeUD_3741 := [[497.37, -11.1, 177.84], [0.129139, 0.695214, 0.685192, -0.174676], [0,0,0,0], [9E9, 9E9, 9E9, 9E9, 9E9, 9E9]];
	VAR robtarget OpenholeUD_3742 := [[493.38, -11.1, 178.14], [0.117647, 0.697251, 0.687831, -0.163978], [0,0,0,0], [9E9, 9E9, 9E9, 9E9, 9E9, 9E9]];
	VAR robtarget OpenholeUD_3743 := [[489.39, -11.1, 178.45], [0.105824, 0.699143, 0.690374, -0.152917], [0,0,0,0], [9E9, 9E9, 9E9, 9E9, 9E9, 9E9]];
	VAR robtarget OpenholeUD_3744 := [[485.4, -11.1, 178.75], [0.093683, 0.700873, 0.692804, -0.141502], [0,0,0,0], [9E9, 9E9, 9E9, 9E9, 9E9, 9E9]];
	VAR robtarget OpenholeUD_3745 := [[481.41, -11.1, 179.05], [0.081247, 0.702424, 0.695101, -0.129748], [0,0,0,0], [9E9, 9E9, 9E9, 9E9, 9E9, 9E9]];
	VAR robtarget OpenholeUD_3746 := [[477.43, -11.1, 179.36], [0.068539, 0.703777, 0.697247, -0.117671], [0,0,0,0], [9E9, 9E9, 9E9, 9E9, 9E9, 9E9]];
	VAR robtarget OpenholeUD_3747 := [[473.44, -11.1, 179.66], [0.055588, 0.704918, 0.699223, -0.105293], [0,0,0,0], [9E9, 9E9, 9E9, 9E9, 9E9, 9E9]];
	VAR robtarget OpenholeUD_3748 := [[469.45, -11.1, 179.97], [0.042427, 0.705833, 0.701012, -0.092642], [0,0,0,0], [9E9, 9E9, 9E9, 9E9, 9E9, 9E9]];
	VAR robtarget OpenholeUD_3749 := [[465.46, -11.1, 180.27], [0.029091, 0.706508, 0.702596, -0.079746], [0,0,0,0], [9E9, 9E9, 9E9, 9E9, 9E9, 9E9]];
	VAR robtarget OpenholeUD_3750 := [[461.47, -11.1, 180.58], [0.01562, 0.706934, 0.70396, -0.06664], [0,0,0,0], [9E9, 9E9, 9E9, 9E9, 9E9, 9E9]];
	VAR robtarget OpenholeUD_3751 := [[457.48, -11.1, 180.88], [0.002057, 0.707104, 0.70509, -0.053361], [0,0,0,0], [9E9, 9E9, 9E9, 9E9, 9E9, 9E9]];
	VAR robtarget OpenholeUD_3752 := [[453.5, -11.1, 181.18], [-0.011554, 0.707012, 0.705977, -0.03995], [0,0,0,0], [9E9, 9E9, 9E9, 9E9, 9E9, 9E9]];
	VAR robtarget OpenholeUD_3753 := [[449.51, -11.1, 181.49], [-0.025169, 0.706659, 0.706612, -0.026449], [0,0,0,0], [9E9, 9E9, 9E9, 9E9, 9E9, 9E9]];
	VAR robtarget OpenholeUD_3754 := [[445.52, -11.1, 181.79], [-0.038742, 0.706045, 0.706989, -0.012902], [0,0,0,0], [9E9, 9E9, 9E9, 9E9, 9E9, 9E9]];
	VAR robtarget OpenholeUD_3755 := [[441.53, -11.1, 182.1], [-0.052228, 0.705175, 0.707106, 0.000647], [0,0,0,0], [9E9, 9E9, 9E9, 9E9, 9E9, 9E9]];
	VAR robtarget OpenholeUD_3756 := [[437.54, -11.1, 182.4], [-0.065583, 0.704059, 0.706965, 0.014152], [0,0,0,0], [9E9, 9E9, 9E9, 9E9, 9E9, 9E9]];
	VAR robtarget OpenholeUD_3757 := [[433.55, -11.1, 182.71], [-0.078766, 0.702706, 0.706569, 0.027571], [0,0,0,0], [9E9, 9E9, 9E9, 9E9, 9E9, 9E9]];
	VAR robtarget OpenholeUD_3758 := [[429.56, -11.1, 183.01], [-0.091738, 0.701131, 0.705925, 0.040863], [0,0,0,0], [9E9, 9E9, 9E9, 9E9, 9E9, 9E9]];
	VAR robtarget OpenholeUD_3759 := [[425.58, -11.1, 183.32], [-0.104466, 0.699347, 0.705043, 0.053987], [0,0,0,0], [9E9, 9E9, 9E9, 9E9, 9E9, 9E9]];
	VAR robtarget OpenholeUD_3760 := [[421.59, -11.1, 183.62], [-0.116917, 0.697374, 0.703934, 0.066908], [0,0,0,0], [9E9, 9E9, 9E9, 9E9, 9E9, 9E9]];
	VAR robtarget OpenholeUD_3761 := [[417.6, -11.1, 183.92], [-0.129065, 0.695228, 0.702613, 0.079594], [0,0,0,0], [9E9, 9E9, 9E9, 9E9, 9E9, 9E9]];
	VAR robtarget OpenholeUD_3762 := [[413.61, -11.1, 184.23], [-0.140887, 0.692929, 0.701094, 0.092016], [0,0,0,0], [9E9, 9E9, 9E9, 9E9, 9E9, 9E9]];
	VAR robtarget OpenholeUD_3763 := [[409.62, -11.1, 184.53], [-0.152366, 0.690496, 0.699395, 0.104149], [0,0,0,0], [9E9, 9E9, 9E9, 9E9, 9E9, 9E9]];
	VAR robtarget OpenholeUD_3764 := [[405.63, -11.1, 184.84], [-0.163487, 0.687948, 0.697532, 0.115973], [0,0,0,0], [9E9, 9E9, 9E9, 9E9, 9E9, 9E9]];
	VAR robtarget OpenholeUD_3765 := [[401.65, -11.1, 185.14], [-0.174242, 0.685303, 0.695522, 0.12747], [0,0,0,0], [9E9, 9E9, 9E9, 9E9, 9E9, 9E9]];
	VAR robtarget OpenholeUD_3766 := [[397.66, -11.1, 185.45], [-0.184623, 0.682579, 0.693385, 0.138628], [0,0,0,0], [9E9, 9E9, 9E9, 9E9, 9E9, 9E9]];
	VAR robtarget OpenholeUD_3767 := [[393.67, -11.1, 185.75], [-0.194628, 0.679794, 0.691135, 0.149439], [0,0,0,0], [9E9, 9E9, 9E9, 9E9, 9E9, 9E9]];
	VAR robtarget OpenholeUD_3768 := [[389.36, -11.1, 186.08], [-0.205013, 0.676735, 0.6886, 0.160719], [0,0,0,0], [9E9, 9E9, 9E9, 9E9, 9E9, 9E9]];
	VAR robtarget OpenholeUD_3769 := [[385.36, -11.1, 186.09], [-0.183051, 0.683002, 0.683002, 0.183051], [0,0,0,0], [9E9, 9E9, 9E9, 9E9, 9E9, 9E9]];
	VAR robtarget OpenholeUD_3770 := [[381.36, -11.1, 186.1], [-0.183051, 0.683002, 0.683002, 0.183051], [0,0,0,0], [9E9, 9E9, 9E9, 9E9, 9E9, 9E9]];
	VAR robtarget OpenholeUD_3771 := [[377.36, -11.1, 186.12], [-0.183051, 0.683002, 0.683002, 0.183051], [0,0,0,0], [9E9, 9E9, 9E9, 9E9, 9E9, 9E9]];
	VAR robtarget OpenholeUD_3772 := [[373.36, -11.1, 186.13], [-0.183051, 0.683002, 0.683002, 0.183051], [0,0,0,0], [9E9, 9E9, 9E9, 9E9, 9E9, 9E9]];
	VAR robtarget OpenholeUD_3773 := [[369.36, -11.1, 186.14], [-0.183051, 0.683002, 0.683002, 0.183051], [0,0,0,0], [9E9, 9E9, 9E9, 9E9, 9E9, 9E9]];
	VAR robtarget OpenholeUD_3774 := [[369.36, -11.1, 186.14], [-0.183051, 0.683002, 0.683002, 0.183051], [0,0,0,0], [9E9, 9E9, 9E9, 9E9, 9E9, 9E9]];
	VAR robtarget OpenholeUD_3775 := [[369.36, -9.9, 186.83], [-0.183051, 0.683002, 0.683002, 0.183051], [0,0,0,0], [9E9, 9E9, 9E9, 9E9, 9E9, 9E9]];
	VAR robtarget OpenholeUD_3776 := [[373.36, -9.9, 186.82], [-0.183051, 0.683002, 0.683002, 0.183051], [0,0,0,0], [9E9, 9E9, 9E9, 9E9, 9E9, 9E9]];
	VAR robtarget OpenholeUD_3777 := [[377.36, -9.9, 186.81], [-0.183051, 0.683002, 0.683002, 0.183051], [0,0,0,0], [9E9, 9E9, 9E9, 9E9, 9E9, 9E9]];
	VAR robtarget OpenholeUD_3778 := [[381.36, -9.9, 186.8], [-0.183051, 0.683002, 0.683002, 0.183051], [0,0,0,0], [9E9, 9E9, 9E9, 9E9, 9E9, 9E9]];
	VAR robtarget OpenholeUD_3779 := [[385.36, -9.9, 186.78], [-0.183051, 0.683002, 0.683002, 0.183051], [0,0,0,0], [9E9, 9E9, 9E9, 9E9, 9E9, 9E9]];
	VAR robtarget OpenholeUD_3780 := [[389.36, -9.9, 186.77], [-0.208383, 0.675704, 0.68939, 0.157294], [0,0,0,0], [9E9, 9E9, 9E9, 9E9, 9E9, 9E9]];
	VAR robtarget OpenholeUD_3781 := [[393.35, -9.9, 186.42], [-0.198862, 0.678568, 0.691699, 0.146808], [0,0,0,0], [9E9, 9E9, 9E9, 9E9, 9E9, 9E9]];
	VAR robtarget OpenholeUD_3782 := [[397.33, -9.9, 186.07], [-0.188965, 0.68139, 0.693911, 0.13597], [0,0,0,0], [9E9, 9E9, 9E9, 9E9, 9E9, 9E9]];
	VAR robtarget OpenholeUD_3783 := [[401.32, -9.9, 185.72], [-0.178692, 0.684156, 0.696009, 0.124786], [0,0,0,0], [9E9, 9E9, 9E9, 9E9, 9E9, 9E9]];
	VAR robtarget OpenholeUD_3784 := [[405.3, -9.9, 185.37], [-0.168043, 0.686849, 0.697976, 0.113265], [0,0,0,0], [9E9, 9E9, 9E9, 9E9, 9E9, 9E9]];
	VAR robtarget OpenholeUD_3785 := [[409.29, -9.9, 185.02], [-0.157025, 0.689451, 0.699796, 0.101421], [0,0,0,0], [9E9, 9E9, 9E9, 9E9, 9E9, 9E9]];
	VAR robtarget OpenholeUD_3786 := [[413.27, -9.9, 184.67], [-0.145646, 0.691944, 0.701449, 0.08927], [0,0,0,0], [9E9, 9E9, 9E9, 9E9, 9E9, 9E9]];
	VAR robtarget OpenholeUD_3787 := [[417.26, -9.9, 184.32], [-0.133919, 0.694309, 0.70292, 0.076833], [0,0,0,0], [9E9, 9E9, 9E9, 9E9, 9E9, 9E9]];
	VAR robtarget OpenholeUD_3788 := [[421.24, -9.9, 183.97], [-0.121861, 0.696527, 0.704192, 0.064134], [0,0,0,0], [9E9, 9E9, 9E9, 9E9, 9E9, 9E9]];
	VAR robtarget OpenholeUD_3789 := [[425.22, -9.9, 183.62], [-0.109494, 0.698578, 0.705251, 0.051203], [0,0,0,0], [9E9, 9E9, 9E9, 9E9, 9E9, 9E9]];
	VAR robtarget OpenholeUD_3790 := [[429.21, -9.9, 183.27], [-0.096842, 0.700444, 0.706081, 0.038072], [0,0,0,0], [9E9, 9E9, 9E9, 9E9, 9E9, 9E9]];
	VAR robtarget OpenholeUD_3791 := [[433.19, -9.9, 182.92], [-0.083937, 0.702107, 0.706673, 0.024777], [0,0,0,0], [9E9, 9E9, 9E9, 9E9, 9E9, 9E9]];
	VAR robtarget OpenholeUD_3792 := [[437.18, -9.9, 182.57], [-0.070812, 0.703552, 0.707016, 0.011357], [0,0,0,0], [9E9, 9E9, 9E9, 9E9, 9E9, 9E9]];
	VAR robtarget OpenholeUD_3793 := [[441.16, -9.9, 182.22], [-0.057505, 0.704765, 0.707104, -0.002145], [0,0,0,0], [9E9, 9E9, 9E9, 9E9, 9E9, 9E9]];
	VAR robtarget OpenholeUD_3794 := [[445.15, -9.9, 181.87], [-0.044056, 0.705733, 0.706933, -0.015688], [0,0,0,0], [9E9, 9E9, 9E9, 9E9, 9E9, 9E9]];
	VAR robtarget OpenholeUD_3795 := [[449.13, -9.9, 181.52], [-0.030509, 0.706448, 0.706503, -0.029226], [0,0,0,0], [9E9, 9E9, 9E9, 9E9, 9E9, 9E9]];
	VAR robtarget OpenholeUD_3796 := [[453.12, -9.9, 181.17], [-0.016908, 0.706905, 0.705815, -0.042714], [0,0,0,0], [9E9, 9E9, 9E9, 9E9, 9E9, 9E9]];
	VAR robtarget OpenholeUD_3797 := [[457.1, -9.9, 180.82], [-0.003299, 0.707099, 0.704877, -0.05611], [0,0,0,0], [9E9, 9E9, 9E9, 9E9, 9E9, 9E9]];
	VAR robtarget OpenholeUD_3798 := [[461.09, -9.9, 180.47], [0.010273, 0.707032, 0.703696, -0.069371], [0,0,0,0], [9E9, 9E9, 9E9, 9E9, 9E9, 9E9]];
	VAR robtarget OpenholeUD_3799 := [[465.07, -9.9, 180.12], [0.023765, 0.706707, 0.702283, -0.082456], [0,0,0,0], [9E9, 9E9, 9E9, 9E9, 9E9, 9E9]];
	VAR robtarget OpenholeUD_3800 := [[469.06, -9.9, 179.77], [0.037132, 0.706131, 0.700651, -0.095329], [0,0,0,0], [9E9, 9E9, 9E9, 9E9, 9E9, 9E9]];
	VAR robtarget OpenholeUD_3801 := [[473.04, -9.9, 179.42], [0.050336, 0.705313, 0.698817, -0.107955], [0,0,0,0], [9E9, 9E9, 9E9, 9E9, 9E9, 9E9]];
	VAR robtarget OpenholeUD_3802 := [[477.03, -9.9, 179.07], [0.063338, 0.704264, 0.696798, -0.120304], [0,0,0,0], [9E9, 9E9, 9E9, 9E9, 9E9, 9E9]];
	VAR robtarget OpenholeUD_3803 := [[481.01, -9.9, 178.72], [0.076107, 0.702999, 0.69461, -0.132351], [0,0,0,0], [9E9, 9E9, 9E9, 9E9, 9E9, 9E9]];
	VAR robtarget OpenholeUD_3804 := [[484.99, -9.9, 178.37], [0.088612, 0.701533, 0.692273, -0.144074], [0,0,0,0], [9E9, 9E9, 9E9, 9E9, 9E9, 9E9]];
	VAR robtarget OpenholeUD_3805 := [[488.98, -9.9, 178.02], [0.100828, 0.699881, 0.689807, -0.155456], [0,0,0,0], [9E9, 9E9, 9E9, 9E9, 9E9, 9E9]];
	VAR robtarget OpenholeUD_3806 := [[492.96, -9.9, 177.67], [0.112733, 0.698062, 0.687229, -0.166482], [0,0,0,0], [9E9, 9E9, 9E9, 9E9, 9E9, 9E9]];
	VAR robtarget OpenholeUD_3807 := [[496.95, -9.9, 177.32], [0.124311, 0.696094, 0.684558, -0.177145], [0,0,0,0], [9E9, 9E9, 9E9, 9E9, 9E9, 9E9]];
	VAR robtarget OpenholeUD_3808 := [[500.93, -9.9, 176.97], [0.135549, 0.693993, 0.681812, -0.187437], [0,0,0,0], [9E9, 9E9, 9E9, 9E9, 9E9, 9E9]];
	VAR robtarget OpenholeUD_3809 := [[504.92, -9.9, 176.62], [0.146437, 0.691778, 0.679007, -0.197357], [0,0,0,0], [9E9, 9E9, 9E9, 9E9, 9E9, 9E9]];
	VAR robtarget OpenholeUD_3810 := [[509.33, -9.9, 176.23], [0.183051, 0.683002, 0.683002, -0.183051], [0,0,0,0], [9E9, 9E9, 9E9, 9E9, 9E9, 9E9]];
	VAR robtarget OpenholeUD_3811 := [[513.33, -9.9, 176.22], [0.183051, 0.683002, 0.683002, -0.183051], [0,0,0,0], [9E9, 9E9, 9E9, 9E9, 9E9, 9E9]];
	VAR robtarget OpenholeUD_3812 := [[517.33, -9.9, 176.21], [0.183051, 0.683002, 0.683002, -0.183051], [0,0,0,0], [9E9, 9E9, 9E9, 9E9, 9E9, 9E9]];
	VAR robtarget OpenholeUD_3813 := [[521.33, -9.9, 176.19], [0.183051, 0.683002, 0.683002, -0.183051], [0,0,0,0], [9E9, 9E9, 9E9, 9E9, 9E9, 9E9]];
	VAR robtarget OpenholeUD_3814 := [[525.33, -9.9, 176.18], [0.183051, 0.683002, 0.683002, -0.183051], [0,0,0,0], [9E9, 9E9, 9E9, 9E9, 9E9, 9E9]];
	VAR robtarget OpenholeUD_3815 := [[529.33, -9.9, 176.17], [0.183051, 0.683002, 0.683002, -0.183051], [0,0,0,0], [9E9, 9E9, 9E9, 9E9, 9E9, 9E9]];
	VAR robtarget OpenholeUD_3816 := [[529.33, -9.9, 176.17], [0.183051, 0.683002, 0.683002, -0.183051], [0,0,0,0], [9E9, 9E9, 9E9, 9E9, 9E9, 9E9]];
	VAR robtarget OpenholeUD_3817 := [[529.33, -8.7, 175.48], [0.183051, 0.683002, 0.683002, -0.183051], [0,0,0,0], [9E9, 9E9, 9E9, 9E9, 9E9, 9E9]];
	VAR robtarget OpenholeUD_3818 := [[525.33, -8.7, 175.49], [0.183051, 0.683002, 0.683002, -0.183051], [0,0,0,0], [9E9, 9E9, 9E9, 9E9, 9E9, 9E9]];
	VAR robtarget OpenholeUD_3819 := [[521.33, -8.7, 175.5], [0.183051, 0.683002, 0.683002, -0.183051], [0,0,0,0], [9E9, 9E9, 9E9, 9E9, 9E9, 9E9]];
	VAR robtarget OpenholeUD_3820 := [[517.33, -8.7, 175.51], [0.183051, 0.683002, 0.683002, -0.183051], [0,0,0,0], [9E9, 9E9, 9E9, 9E9, 9E9, 9E9]];
	VAR robtarget OpenholeUD_3821 := [[513.33, -8.7, 175.53], [0.183051, 0.683002, 0.683002, -0.183051], [0,0,0,0], [9E9, 9E9, 9E9, 9E9, 9E9, 9E9]];
	VAR robtarget OpenholeUD_3822 := [[509.33, -8.7, 175.54], [0.183051, 0.683002, 0.683002, -0.183051], [0,0,0,0], [9E9, 9E9, 9E9, 9E9, 9E9, 9E9]];
	VAR robtarget OpenholeUD_3823 := [[505.35, -8.7, 175.93], [0.144095, 0.692269, 0.677691, -0.20183], [0,0,0,0], [9E9, 9E9, 9E9, 9E9, 9E9, 9E9]];
	VAR robtarget OpenholeUD_3824 := [[501.37, -8.7, 176.33], [0.13319, 0.69445, 0.680533, -0.192028], [0,0,0,0], [9E9, 9E9, 9E9, 9E9, 9E9, 9E9]];
	VAR robtarget OpenholeUD_3825 := [[497.39, -8.7, 176.73], [0.121938, 0.696514, 0.683322, -0.181853], [0,0,0,0], [9E9, 9E9, 9E9, 9E9, 9E9, 9E9]];
	VAR robtarget OpenholeUD_3826 := [[493.41, -8.7, 177.12], [0.110347, 0.698444, 0.686042, -0.171307], [0,0,0,0], [9E9, 9E9, 9E9, 9E9, 9E9, 9E9]];
	VAR robtarget OpenholeUD_3827 := [[489.43, -8.7, 177.52], [0.098431, 0.700222, 0.688675, -0.160394], [0,0,0,0], [9E9, 9E9, 9E9, 9E9, 9E9, 9E9]];
	VAR robtarget OpenholeUD_3828 := [[485.45, -8.7, 177.91], [0.086207, 0.701832, 0.691204, -0.149122], [0,0,0,0], [9E9, 9E9, 9E9, 9E9, 9E9, 9E9]];
	VAR robtarget OpenholeUD_3829 := [[481.47, -8.7, 178.31], [0.073696, 0.703256, 0.693608, -0.137505], [0,0,0,0], [9E9, 9E9, 9E9, 9E9, 9E9, 9E9]];
	VAR robtarget OpenholeUD_3830 := [[477.49, -8.7, 178.7], [0.060923, 0.704477, 0.69587, -0.125557], [0,0,0,0], [9E9, 9E9, 9E9, 9E9, 9E9, 9E9]];
	VAR robtarget OpenholeUD_3831 := [[473.5, -8.7, 179.1], [0.047918, 0.705481, 0.697971, -0.1133], [0,0,0,0], [9E9, 9E9, 9E9, 9E9, 9E9, 9E9]];
	VAR robtarget OpenholeUD_3832 := [[469.52, -8.7, 179.5], [0.034715, 0.706254, 0.699891, -0.100758], [0,0,0,0], [9E9, 9E9, 9E9, 9E9, 9E9, 9E9]];
	VAR robtarget OpenholeUD_3833 := [[465.54, -8.7, 179.89], [0.02135, 0.706784, 0.701614, -0.087961], [0,0,0,0], [9E9, 9E9, 9E9, 9E9, 9E9, 9E9]];
	VAR robtarget OpenholeUD_3834 := [[461.56, -8.7, 180.29], [0.007863, 0.707063, 0.703124, -0.074941], [0,0,0,0], [9E9, 9E9, 9E9, 9E9, 9E9, 9E9]];
	VAR robtarget OpenholeUD_3835 := [[457.58, -8.7, 180.68], [-0.005703, 0.707084, 0.704407, -0.061735], [0,0,0,0], [9E9, 9E9, 9E9, 9E9, 9E9, 9E9]];
	VAR robtarget OpenholeUD_3836 := [[453.6, -8.7, 181.08], [-0.019304, 0.706843, 0.70545, -0.048382], [0,0,0,0], [9E9, 9E9, 9E9, 9E9, 9E9, 9E9]];
	VAR robtarget OpenholeUD_3837 := [[449.62, -8.7, 181.47], [-0.032895, 0.706341, 0.706244, -0.034924], [0,0,0,0], [9E9, 9E9, 9E9, 9E9, 9E9, 9E9]];
	VAR robtarget OpenholeUD_3838 := [[445.64, -8.7, 181.87], [-0.04643, 0.705581, 0.706783, -0.021404], [0,0,0,0], [9E9, 9E9, 9E9, 9E9, 9E9, 9E9]];
	VAR robtarget OpenholeUD_3839 := [[441.66, -8.7, 182.27], [-0.059866, 0.704568, 0.707063, -0.007867], [0,0,0,0], [9E9, 9E9, 9E9, 9E9, 9E9, 9E9]];
	VAR robtarget OpenholeUD_3840 := [[437.68, -8.7, 182.66], [-0.073158, 0.703312, 0.707084, 0.005643], [0,0,0,0], [9E9, 9E9, 9E9, 9E9, 9E9, 9E9]];
	VAR robtarget OpenholeUD_3841 := [[433.7, -8.7, 183.06], [-0.086267, 0.701825, 0.706849, 0.019083], [0,0,0,0], [9E9, 9E9, 9E9, 9E9, 9E9, 9E9]];
	VAR robtarget OpenholeUD_3842 := [[429.72, -8.7, 183.45], [-0.099154, 0.70012, 0.706364, 0.03241], [0,0,0,0], [9E9, 9E9, 9E9, 9E9, 9E9, 9E9]];
	VAR robtarget OpenholeUD_3843 := [[425.74, -8.7, 183.85], [-0.111786, 0.698215, 0.705636, 0.045584], [0,0,0,0], [9E9, 9E9, 9E9, 9E9, 9E9, 9E9]];
	VAR robtarget OpenholeUD_3844 := [[421.76, -8.7, 184.24], [-0.124134, 0.696126, 0.704677, 0.058569], [0,0,0,0], [9E9, 9E9, 9E9, 9E9, 9E9, 9E9]];
	VAR robtarget OpenholeUD_3845 := [[417.78, -8.7, 184.64], [-0.13617, 0.693872, 0.7035, 0.071332], [0,0,0,0], [9E9, 9E9, 9E9, 9E9, 9E9, 9E9]];
	VAR robtarget OpenholeUD_3846 := [[413.8, -8.7, 185.04], [-0.147874, 0.691472, 0.702119, 0.083842], [0,0,0,0], [9E9, 9E9, 9E9, 9E9, 9E9, 9E9]];
	VAR robtarget OpenholeUD_3847 := [[409.82, -8.7, 185.43], [-0.15923, 0.688945, 0.70055, 0.096073], [0,0,0,0], [9E9, 9E9, 9E9, 9E9, 9E9, 9E9]];
	VAR robtarget OpenholeUD_3848 := [[405.84, -8.7, 185.83], [-0.170223, 0.686312, 0.69881, 0.108005], [0,0,0,0], [9E9, 9E9, 9E9, 9E9, 9E9, 9E9]];
	VAR robtarget OpenholeUD_3849 := [[401.86, -8.7, 186.22], [-0.180846, 0.68359, 0.696916, 0.119618], [0,0,0,0], [9E9, 9E9, 9E9, 9E9, 9E9, 9E9]];
	VAR robtarget OpenholeUD_3850 := [[397.88, -8.7, 186.62], [-0.191093, 0.680796, 0.694885, 0.130899], [0,0,0,0], [9E9, 9E9, 9E9, 9E9, 9E9, 9E9]];
	VAR robtarget OpenholeUD_3851 := [[393.9, -8.7, 187.01], [-0.200963, 0.677948, 0.692735, 0.141839], [0,0,0,0], [9E9, 9E9, 9E9, 9E9, 9E9, 9E9]];
	VAR robtarget OpenholeUD_3852 := [[389.37, -8.7, 187.46], [-0.211743, 0.674659, 0.690162, 0.15387], [0,0,0,0], [9E9, 9E9, 9E9, 9E9, 9E9, 9E9]];
	VAR robtarget OpenholeUD_3853 := [[385.37, -8.7, 187.48], [-0.183051, 0.683002, 0.683002, 0.183051], [0,0,0,0], [9E9, 9E9, 9E9, 9E9, 9E9, 9E9]];
	VAR robtarget OpenholeUD_3854 := [[381.37, -8.7, 187.49], [-0.183051, 0.683002, 0.683002, 0.183051], [0,0,0,0], [9E9, 9E9, 9E9, 9E9, 9E9, 9E9]];
	VAR robtarget OpenholeUD_3855 := [[377.37, -8.7, 187.5], [-0.183051, 0.683002, 0.683002, 0.183051], [0,0,0,0], [9E9, 9E9, 9E9, 9E9, 9E9, 9E9]];
	VAR robtarget OpenholeUD_3856 := [[373.37, -8.7, 187.52], [-0.183051, 0.683002, 0.683002, 0.183051], [0,0,0,0], [9E9, 9E9, 9E9, 9E9, 9E9, 9E9]];
	VAR robtarget OpenholeUD_3857 := [[369.37, -8.7, 187.53], [-0.183051, 0.683002, 0.683002, 0.183051], [0,0,0,0], [9E9, 9E9, 9E9, 9E9, 9E9, 9E9]];
	VAR robtarget OpenholeUD_3858 := [[369.37, -8.7, 187.53], [-0.183051, 0.683002, 0.683002, 0.183051], [0,0,0,0], [9E9, 9E9, 9E9, 9E9, 9E9, 9E9]];
	VAR robtarget OpenholeUD_3859 := [[369.37, -7.5, 188.22], [-0.183051, 0.683002, 0.683002, 0.183051], [0,0,0,0], [9E9, 9E9, 9E9, 9E9, 9E9, 9E9]];
	VAR robtarget OpenholeUD_3860 := [[373.37, -7.5, 188.21], [-0.183051, 0.683002, 0.683002, 0.183051], [0,0,0,0], [9E9, 9E9, 9E9, 9E9, 9E9, 9E9]];
	VAR robtarget OpenholeUD_3861 := [[377.37, -7.5, 188.2], [-0.183051, 0.683002, 0.683002, 0.183051], [0,0,0,0], [9E9, 9E9, 9E9, 9E9, 9E9, 9E9]];
	VAR robtarget OpenholeUD_3862 := [[381.37, -7.5, 188.18], [-0.183051, 0.683002, 0.683002, 0.183051], [0,0,0,0], [9E9, 9E9, 9E9, 9E9, 9E9, 9E9]];
	VAR robtarget OpenholeUD_3863 := [[385.37, -7.5, 188.17], [-0.183051, 0.683002, 0.683002, 0.183051], [0,0,0,0], [9E9, 9E9, 9E9, 9E9, 9E9, 9E9]];
	VAR robtarget OpenholeUD_3864 := [[389.37, -7.5, 188.16], [-0.215092, 0.673599, 0.690916, 0.150448], [0,0,0,0], [9E9, 9E9, 9E9, 9E9, 9E9, 9E9]];
	VAR robtarget OpenholeUD_3865 := [[393.34, -7.5, 187.72], [-0.205731, 0.676517, 0.693139, 0.139853], [0,0,0,0], [9E9, 9E9, 9E9, 9E9, 9E9, 9E9]];
	VAR robtarget OpenholeUD_3866 := [[397.32, -7.5, 187.28], [-0.195993, 0.679402, 0.695257, 0.12891], [0,0,0,0], [9E9, 9E9, 9E9, 9E9, 9E9, 9E9]];
	VAR robtarget OpenholeUD_3867 := [[401.29, -7.5, 186.83], [-0.185878, 0.682238, 0.697255, 0.117627], [0,0,0,0], [9E9, 9E9, 9E9, 9E9, 9E9, 9E9]];
	VAR robtarget OpenholeUD_3868 := [[405.27, -7.5, 186.39], [-0.175386, 0.685011, 0.699115, 0.106013], [0,0,0,0], [9E9, 9E9, 9E9, 9E9, 9E9, 9E9]];
	VAR robtarget OpenholeUD_3869 := [[409.25, -7.5, 185.95], [-0.164521, 0.687701, 0.70082, 0.094083], [0,0,0,0], [9E9, 9E9, 9E9, 9E9, 9E9, 9E9]];
	VAR robtarget OpenholeUD_3870 := [[413.22, -7.5, 185.51], [-0.15329, 0.690291, 0.702353, 0.081854], [0,0,0,0], [9E9, 9E9, 9E9, 9E9, 9E9, 9E9]];
	VAR robtarget OpenholeUD_3871 := [[417.2, -7.5, 185.07], [-0.141705, 0.692762, 0.703698, 0.069349], [0,0,0,0], [9E9, 9E9, 9E9, 9E9, 9E9, 9E9]];
	VAR robtarget OpenholeUD_3872 := [[421.17, -7.5, 184.63], [-0.129781, 0.695095, 0.704839, 0.056592], [0,0,0,0], [9E9, 9E9, 9E9, 9E9, 9E9, 9E9]];
	VAR robtarget OpenholeUD_3873 := [[425.15, -7.5, 184.19], [-0.11754, 0.697269, 0.705761, 0.043613], [0,0,0,0], [9E9, 9E9, 9E9, 9E9, 9E9, 9E9]];
	VAR robtarget OpenholeUD_3874 := [[429.12, -7.5, 183.75], [-0.105004, 0.699267, 0.706451, 0.030446], [0,0,0,0], [9E9, 9E9, 9E9, 9E9, 9E9, 9E9]];
	VAR robtarget OpenholeUD_3875 := [[433.1, -7.5, 183.3], [-0.092204, 0.70107, 0.706899, 0.017127], [0,0,0,0], [9E9, 9E9, 9E9, 9E9, 9E9, 9E9]];
	VAR robtarget OpenholeUD_3876 := [[437.07, -7.5, 182.86], [-0.079171, 0.702661, 0.707097, 0.003696], [0,0,0,0], [9E9, 9E9, 9E9, 9E9, 9E9, 9E9]];
	VAR robtarget OpenholeUD_3877 := [[441.05, -7.5, 182.42], [-0.065942, 0.704025, 0.707039, -0.009805], [0,0,0,0], [9E9, 9E9, 9E9, 9E9, 9E9, 9E9]];
	VAR robtarget OpenholeUD_3878 := [[445.03, -7.5, 181.98], [-0.052558, 0.705151, 0.706722, -0.023332], [0,0,0,0], [9E9, 9E9, 9E9, 9E9, 9E9, 9E9]];
	VAR robtarget OpenholeUD_3879 := [[449, -7.5, 181.54], [-0.039059, 0.706027, 0.706146, -0.036842], [0,0,0,0], [9E9, 9E9, 9E9, 9E9, 9E9, 9E9]];
	VAR robtarget OpenholeUD_3880 := [[452.98, -7.5, 181.1], [-0.025491, 0.706647, 0.705316, -0.050291], [0,0,0,0], [9E9, 9E9, 9E9, 9E9, 9E9, 9E9]];
	VAR robtarget OpenholeUD_3881 := [[456.95, -7.5, 180.66], [-0.011898, 0.707007, 0.704238, -0.063634], [0,0,0,0], [9E9, 9E9, 9E9, 9E9, 9E9, 9E9]];
	VAR robtarget OpenholeUD_3882 := [[460.93, -7.5, 180.22], [0.001675, 0.707105, 0.70292, -0.07683], [0,0,0,0], [9E9, 9E9, 9E9, 9E9, 9E9, 9E9]];
	VAR robtarget OpenholeUD_3883 := [[464.9, -7.5, 179.77], [0.015182, 0.706944, 0.701376, -0.089839], [0,0,0,0], [9E9, 9E9, 9E9, 9E9, 9E9, 9E9]];
	VAR robtarget OpenholeUD_3884 := [[468.88, -7.5, 179.33], [0.028581, 0.706529, 0.69962, -0.102626], [0,0,0,0], [9E9, 9E9, 9E9, 9E9, 9E9, 9E9]];
	VAR robtarget OpenholeUD_3885 := [[472.85, -7.5, 178.89], [0.041832, 0.705868, 0.697667, -0.115157], [0,0,0,0], [9E9, 9E9, 9E9, 9E9, 9E9, 9E9]];
	VAR robtarget OpenholeUD_3886 := [[476.83, -7.5, 178.45], [0.054896, 0.704973, 0.695535, -0.127403], [0,0,0,0], [9E9, 9E9, 9E9, 9E9, 9E9, 9E9]];
	VAR robtarget OpenholeUD_3887 := [[480.81, -7.5, 178.01], [0.067739, 0.703855, 0.693242, -0.139339], [0,0,0,0], [9E9, 9E9, 9E9, 9E9, 9E9, 9E9]];
	VAR robtarget OpenholeUD_3888 := [[484.78, -7.5, 177.57], [0.08033, 0.702529, 0.690808, -0.150945], [0,0,0,0], [9E9, 9E9, 9E9, 9E9, 9E9, 9E9]];
	VAR robtarget OpenholeUD_3889 := [[488.76, -7.5, 177.13], [0.092643, 0.701012, 0.688251, -0.162205], [0,0,0,0], [9E9, 9E9, 9E9, 9E9, 9E9, 9E9]];
	VAR robtarget OpenholeUD_3890 := [[492.73, -7.5, 176.69], [0.104656, 0.699319, 0.685591, -0.173105], [0,0,0,0], [9E9, 9E9, 9E9, 9E9, 9E9, 9E9]];
	VAR robtarget OpenholeUD_3891 := [[496.71, -7.5, 176.25], [0.11635, 0.697469, 0.682845, -0.183638], [0,0,0,0], [9E9, 9E9, 9E9, 9E9, 9E9, 9E9]];
	VAR robtarget OpenholeUD_3892 := [[500.68, -7.5, 175.8], [0.127711, 0.695478, 0.680031, -0.193799], [0,0,0,0], [9E9, 9E9, 9E9, 9E9, 9E9, 9E9]];
	VAR robtarget OpenholeUD_3893 := [[504.66, -7.5, 175.36], [0.138728, 0.693365, 0.677165, -0.203586], [0,0,0,0], [9E9, 9E9, 9E9, 9E9, 9E9, 9E9]];
	VAR robtarget OpenholeUD_3894 := [[509.33, -7.5, 174.84], [0.183051, 0.683002, 0.683002, -0.183051], [0,0,0,0], [9E9, 9E9, 9E9, 9E9, 9E9, 9E9]];
	VAR robtarget OpenholeUD_3895 := [[513.33, -7.5, 174.83], [0.183051, 0.683002, 0.683002, -0.183051], [0,0,0,0], [9E9, 9E9, 9E9, 9E9, 9E9, 9E9]];
	VAR robtarget OpenholeUD_3896 := [[517.33, -7.5, 174.82], [0.183051, 0.683002, 0.683002, -0.183051], [0,0,0,0], [9E9, 9E9, 9E9, 9E9, 9E9, 9E9]];
	VAR robtarget OpenholeUD_3897 := [[521.33, -7.5, 174.81], [0.183051, 0.683002, 0.683002, -0.183051], [0,0,0,0], [9E9, 9E9, 9E9, 9E9, 9E9, 9E9]];
	VAR robtarget OpenholeUD_3898 := [[529.33, -7.5, 174.78], [0.183051, 0.683002, 0.683002, -0.183051], [0,0,0,0], [9E9, 9E9, 9E9, 9E9, 9E9, 9E9]];
	VAR robtarget OpenholeUD_3899 := [[529.33, -7.5, 174.78], [0.183051, 0.683002, 0.683002, -0.183051], [0,0,0,0], [9E9, 9E9, 9E9, 9E9, 9E9, 9E9]];
	VAR robtarget OpenholeUD_3900 := [[529.32, -6.3, 174.09], [0.183051, 0.683002, 0.683002, -0.183051], [0,0,0,0], [9E9, 9E9, 9E9, 9E9, 9E9, 9E9]];
	VAR robtarget OpenholeUD_3901 := [[525.32, -6.3, 174.1], [0.183051, 0.683002, 0.683002, -0.183051], [0,0,0,0], [9E9, 9E9, 9E9, 9E9, 9E9, 9E9]];
	VAR robtarget OpenholeUD_3902 := [[521.32, -6.3, 174.11], [0.183051, 0.683002, 0.683002, -0.183051], [0,0,0,0], [9E9, 9E9, 9E9, 9E9, 9E9, 9E9]];
	VAR robtarget OpenholeUD_3903 := [[517.32, -6.3, 174.13], [0.183051, 0.683002, 0.683002, -0.183051], [0,0,0,0], [9E9, 9E9, 9E9, 9E9, 9E9, 9E9]];
	VAR robtarget OpenholeUD_3904 := [[509.32, -6.3, 174.15], [0.183051, 0.683002, 0.683002, -0.183051], [0,0,0,0], [9E9, 9E9, 9E9, 9E9, 9E9, 9E9]];
	VAR robtarget OpenholeUD_3905 := [[505.35, -6.3, 174.64], [0.137125, 0.693683, 0.67562, -0.208657], [0,0,0,0], [9E9, 9E9, 9E9, 9E9, 9E9, 9E9]];
	VAR robtarget OpenholeUD_3906 := [[501.38, -6.3, 175.12], [0.126118, 0.695769, 0.678522, -0.199016], [0,0,0,0], [9E9, 9E9, 9E9, 9E9, 9E9, 9E9]];
	VAR robtarget OpenholeUD_3907 := [[497.41, -6.3, 175.61], [0.114769, 0.697731, 0.68138, -0.189], [0,0,0,0], [9E9, 9E9, 9E9, 9E9, 9E9, 9E9]];
	VAR robtarget OpenholeUD_3908 := [[493.44, -6.3, 176.1], [0.103088, 0.699552, 0.684177, -0.178611], [0,0,0,0], [9E9, 9E9, 9E9, 9E9, 9E9, 9E9]];
	VAR robtarget OpenholeUD_3909 := [[489.47, -6.3, 176.58], [0.091089, 0.701215, 0.686896, -0.167851], [0,0,0,0], [9E9, 9E9, 9E9, 9E9, 9E9, 9E9]];
	VAR robtarget OpenholeUD_3910 := [[485.5, -6.3, 177.07], [0.078791, 0.702703, 0.689519, -0.156728], [0,0,0,0], [9E9, 9E9, 9E9, 9E9, 9E9, 9E9]];
	VAR robtarget OpenholeUD_3911 := [[481.53, -6.3, 177.56], [0.066214, 0.704, 0.692027, -0.145254], [0,0,0,0], [9E9, 9E9, 9E9, 9E9, 9E9, 9E9]];
	VAR robtarget OpenholeUD_3912 := [[477.56, -6.3, 178.04], [0.053387, 0.705089, 0.694401, -0.133443], [0,0,0,0], [9E9, 9E9, 9E9, 9E9, 9E9, 9E9]];
	VAR robtarget OpenholeUD_3913 := [[473.59, -6.3, 178.53], [0.040339, 0.705955, 0.696623, -0.121314], [0,0,0,0], [9E9, 9E9, 9E9, 9E9, 9E9, 9E9]];
	VAR robtarget OpenholeUD_3914 := [[469.62, -6.3, 179.02], [0.027103, 0.706587, 0.698672, -0.108891], [0,0,0,0], [9E9, 9E9, 9E9, 9E9, 9E9, 9E9]];
	VAR robtarget OpenholeUD_3915 := [[465.65, -6.3, 179.5], [0.013718, 0.706974, 0.700532, -0.096201], [0,0,0,0], [9E9, 9E9, 9E9, 9E9, 9E9, 9E9]];
	VAR robtarget OpenholeUD_3916 := [[461.68, -6.3, 179.99], [0.000225, 0.707107, 0.702186, -0.083277], [0,0,0,0], [9E9, 9E9, 9E9, 9E9, 9E9, 9E9]];
	VAR robtarget OpenholeUD_3917 := [[457.71, -6.3, 180.48], [-0.013336, 0.706981, 0.703618, -0.070152], [0,0,0,0], [9E9, 9E9, 9E9, 9E9, 9E9, 9E9]];
	VAR robtarget OpenholeUD_3918 := [[453.74, -6.3, 180.96], [-0.026918, 0.706594, 0.704816, -0.056867], [0,0,0,0], [9E9, 9E9, 9E9, 9E9, 9E9, 9E9]];
	VAR robtarget OpenholeUD_3919 := [[449.77, -6.3, 181.45], [-0.040477, 0.705947, 0.70577, -0.043462], [0,0,0,0], [9E9, 9E9, 9E9, 9E9, 9E9, 9E9]];
	VAR robtarget OpenholeUD_3920 := [[445.8, -6.3, 181.94], [-0.053967, 0.705044, 0.706471, -0.029979], [0,0,0,0], [9E9, 9E9, 9E9, 9E9, 9E9, 9E9]];
	VAR robtarget OpenholeUD_3921 := [[441.83, -6.3, 182.42], [-0.067346, 0.703892, 0.706915, -0.016463], [0,0,0,0], [9E9, 9E9, 9E9, 9E9, 9E9, 9E9]];
	VAR robtarget OpenholeUD_3922 := [[437.86, -6.3, 182.91], [-0.08057, 0.702502, 0.707101, -0.002958], [0,0,0,0], [9E9, 9E9, 9E9, 9E9, 9E9, 9E9]];
	VAR robtarget OpenholeUD_3923 := [[433.89, -6.3, 183.4], [-0.093599, 0.700885, 0.707029, 0.010492], [0,0,0,0], [9E9, 9E9, 9E9, 9E9, 9E9, 9E9]];
	VAR robtarget OpenholeUD_3924 := [[429.92, -6.3, 183.88], [-0.106398, 0.699056, 0.706705, 0.023845], [0,0,0,0], [9E9, 9E9, 9E9, 9E9, 9E9, 9E9]];
	VAR robtarget OpenholeUD_3925 := [[425.95, -6.3, 184.37], [-0.118932, 0.697033, 0.706135, 0.037061], [0,0,0,0], [9E9, 9E9, 9E9, 9E9, 9E9, 9E9]];
	VAR robtarget OpenholeUD_3926 := [[421.98, -6.3, 184.86], [-0.131174, 0.694833, 0.70533, 0.050101], [0,0,0,0], [9E9, 9E9, 9E9, 9E9, 9E9, 9E9]];
	VAR robtarget OpenholeUD_3927 := [[418.01, -6.3, 185.34], [-0.143097, 0.692476, 0.704301, 0.062933], [0,0,0,0], [9E9, 9E9, 9E9, 9E9, 9E9, 9E9]];
	VAR robtarget OpenholeUD_3928 := [[414.04, -6.3, 185.83], [-0.154683, 0.689981, 0.703062, 0.075524], [0,0,0,0], [9E9, 9E9, 9E9, 9E9, 9E9, 9E9]];
	VAR robtarget OpenholeUD_3929 := [[410.07, -6.3, 186.31], [-0.165915, 0.687366, 0.701629, 0.087848], [0,0,0,0], [9E9, 9E9, 9E9, 9E9, 9E9, 9E9]];
	VAR robtarget OpenholeUD_3930 := [[406.1, -6.3, 186.8], [-0.176781, 0.684652, 0.700017, 0.099881], [0,0,0,0], [9E9, 9E9, 9E9, 9E9, 9E9, 9E9]];
	VAR robtarget OpenholeUD_3931 := [[402.13, -6.3, 187.29], [-0.187273, 0.681857, 0.698244, 0.111606], [0,0,0,0], [9E9, 9E9, 9E9, 9E9, 9E9, 9E9]];
	VAR robtarget OpenholeUD_3932 := [[398.16, -6.3, 187.77], [-0.197388, 0.678998, 0.696326, 0.123006], [0,0,0,0], [9E9, 9E9, 9E9, 9E9, 9E9, 9E9]];
	VAR robtarget OpenholeUD_3933 := [[394.19, -6.3, 188.26], [-0.207125, 0.676091, 0.69428, 0.13407], [0,0,0,0], [9E9, 9E9, 9E9, 9E9, 9E9, 9E9]];
	VAR robtarget OpenholeUD_3934 := [[389.37, -6.3, 188.85], [-0.218429, 0.672524, 0.691652, 0.147029], [0,0,0,0], [9E9, 9E9, 9E9, 9E9, 9E9, 9E9]];
	VAR robtarget OpenholeUD_3935 := [[385.37, -6.3, 188.86], [-0.183051, 0.683002, 0.683002, 0.183051], [0,0,0,0], [9E9, 9E9, 9E9, 9E9, 9E9, 9E9]];
	VAR robtarget OpenholeUD_3936 := [[381.37, -6.3, 188.88], [-0.183051, 0.683002, 0.683002, 0.183051], [0,0,0,0], [9E9, 9E9, 9E9, 9E9, 9E9, 9E9]];
	VAR robtarget OpenholeUD_3937 := [[377.37, -6.3, 188.89], [-0.183051, 0.683002, 0.683002, 0.183051], [0,0,0,0], [9E9, 9E9, 9E9, 9E9, 9E9, 9E9]];
	VAR robtarget OpenholeUD_3938 := [[373.37, -6.3, 188.9], [-0.183051, 0.683002, 0.683002, 0.183051], [0,0,0,0], [9E9, 9E9, 9E9, 9E9, 9E9, 9E9]];
	VAR robtarget OpenholeUD_3939 := [[369.37, -6.3, 188.91], [-0.183051, 0.683002, 0.683002, 0.183051], [0,0,0,0], [9E9, 9E9, 9E9, 9E9, 9E9, 9E9]];
	VAR robtarget OpenholeUD_3940 := [[369.37, -6.3, 188.91], [-0.183051, 0.683002, 0.683002, 0.183051], [0,0,0,0], [9E9, 9E9, 9E9, 9E9, 9E9, 9E9]];
	VAR robtarget OpenholeUD_3941 := [[369.37, -5.1, 189.61], [-0.183051, 0.683002, 0.683002, 0.183051], [0,0,0,0], [9E9, 9E9, 9E9, 9E9, 9E9, 9E9]];
	VAR robtarget OpenholeUD_3942 := [[373.37, -5.1, 189.59], [-0.183051, 0.683002, 0.683002, 0.183051], [0,0,0,0], [9E9, 9E9, 9E9, 9E9, 9E9, 9E9]];
	VAR robtarget OpenholeUD_3943 := [[377.37, -5.1, 189.58], [-0.183051, 0.683002, 0.683002, 0.183051], [0,0,0,0], [9E9, 9E9, 9E9, 9E9, 9E9, 9E9]];
	VAR robtarget OpenholeUD_3944 := [[381.37, -5.1, 189.57], [-0.183051, 0.683002, 0.683002, 0.183051], [0,0,0,0], [9E9, 9E9, 9E9, 9E9, 9E9, 9E9]];
	VAR robtarget OpenholeUD_3945 := [[385.37, -5.1, 189.56], [-0.183051, 0.683002, 0.683002, 0.183051], [0,0,0,0], [9E9, 9E9, 9E9, 9E9, 9E9, 9E9]];
	VAR robtarget OpenholeUD_3946 := [[389.37, -5.1, 189.54], [-0.221754, 0.671435, 0.692369, 0.143613], [0,0,0,0], [9E9, 9E9, 9E9, 9E9, 9E9, 9E9]];
	VAR robtarget OpenholeUD_3947 := [[393.34, -5.1, 189.01], [-0.212555, 0.674404, 0.694502, 0.132917], [0,0,0,0], [9E9, 9E9, 9E9, 9E9, 9E9, 9E9]];
	VAR robtarget OpenholeUD_3948 := [[397.3, -5.1, 188.48], [-0.202982, 0.677347, 0.696524, 0.121878], [0,0,0,0], [9E9, 9E9, 9E9, 9E9, 9E9, 9E9]];
	VAR robtarget OpenholeUD_3949 := [[401.27, -5.1, 187.95], [-0.193029, 0.68025, 0.698419, 0.110505], [0,0,0,0], [9E9, 9E9, 9E9, 9E9, 9E9, 9E9]];
	VAR robtarget OpenholeUD_3950 := [[405.23, -5.1, 187.42], [-0.182697, 0.683097, 0.700169, 0.098807], [0,0,0,0], [9E9, 9E9, 9E9, 9E9, 9E9, 9E9]];
	VAR robtarget OpenholeUD_3951 := [[409.19, -5.1, 186.89], [-0.17199, 0.685871, 0.701759, 0.086801], [0,0,0,0], [9E9, 9E9, 9E9, 9E9, 9E9, 9E9]];
	VAR robtarget OpenholeUD_3952 := [[413.16, -5.1, 186.35], [-0.160913, 0.688554, 0.703171, 0.074504], [0,0,0,0], [9E9, 9E9, 9E9, 9E9, 9E9, 9E9]];
	VAR robtarget OpenholeUD_3953 := [[417.12, -5.1, 185.82], [-0.149476, 0.691127, 0.704389, 0.06194], [0,0,0,0], [9E9, 9E9, 9E9, 9E9, 9E9, 9E9]];
	VAR robtarget OpenholeUD_3954 := [[421.09, -5.1, 185.29], [-0.137695, 0.693571, 0.705398, 0.049134], [0,0,0,0], [9E9, 9E9, 9E9, 9E9, 9E9, 9E9]];
	VAR robtarget OpenholeUD_3955 := [[425.05, -5.1, 184.76], [-0.125587, 0.695865, 0.706184, 0.036118], [0,0,0,0], [9E9, 9E9, 9E9, 9E9, 9E9, 9E9]];
	VAR robtarget OpenholeUD_3956 := [[429.02, -5.1, 184.23], [-0.113176, 0.697991, 0.706735, 0.022924], [0,0,0,0], [9E9, 9E9, 9E9, 9E9, 9E9, 9E9]];
	VAR robtarget OpenholeUD_3957 := [[432.98, -5.1, 183.7], [-0.100489, 0.69993, 0.707042, 0.009591], [0,0,0,0], [9E9, 9E9, 9E9, 9E9, 9E9, 9E9]];
	VAR robtarget OpenholeUD_3958 := [[436.95, -5.1, 183.16], [-0.087558, 0.701665, 0.707096, -0.003842], [0,0,0,0], [9E9, 9E9, 9E9, 9E9, 9E9, 9E9]];
	VAR robtarget OpenholeUD_3959 := [[440.91, -5.1, 182.63], [-0.074417, 0.70318, 0.706894, -0.017332], [0,0,0,0], [9E9, 9E9, 9E9, 9E9, 9E9, 9E9]];
	VAR robtarget OpenholeUD_3960 := [[444.87, -5.1, 182.1], [-0.061106, 0.704462, 0.706434, -0.030837], [0,0,0,0], [9E9, 9E9, 9E9, 9E9, 9E9, 9E9]];
	VAR robtarget OpenholeUD_3961 := [[448.84, -5.1, 181.57], [-0.047666, 0.705498, 0.705717, -0.044312], [0,0,0,0], [9E9, 9E9, 9E9, 9E9, 9E9, 9E9]];
	VAR robtarget OpenholeUD_3962 := [[452.8, -5.1, 181.04], [-0.034141, 0.706282, 0.704748, -0.057714], [0,0,0,0], [9E9, 9E9, 9E9, 9E9, 9E9, 9E9]];
	VAR robtarget OpenholeUD_3963 := [[456.77, -5.1, 180.51], [-0.020575, 0.706807, 0.703533, -0.070998], [0,0,0,0], [9E9, 9E9, 9E9, 9E9, 9E9, 9E9]];
	VAR robtarget OpenholeUD_3964 := [[460.73, -5.1, 179.97], [-0.007013, 0.707072, 0.702085, -0.084124], [0,0,0,0], [9E9, 9E9, 9E9, 9E9, 9E9, 9E9]];
	VAR robtarget OpenholeUD_3965 := [[464.7, -5.1, 179.44], [0.006501, 0.707077, 0.700415, -0.097054], [0,0,0,0], [9E9, 9E9, 9E9, 9E9, 9E9, 9E9]];
	VAR robtarget OpenholeUD_3966 := [[468.66, -5.1, 178.91], [0.019922, 0.706826, 0.698537, -0.109751], [0,0,0,0], [9E9, 9E9, 9E9, 9E9, 9E9, 9E9]];
	VAR robtarget OpenholeUD_3967 := [[472.63, -5.1, 178.38], [0.03321, 0.706326, 0.69647, -0.122185], [0,0,0,0], [9E9, 9E9, 9E9, 9E9, 9E9, 9E9]];
	VAR robtarget OpenholeUD_3968 := [[476.59, -5.1, 177.85], [0.046327, 0.705588, 0.694231, -0.134325], [0,0,0,0], [9E9, 9E9, 9E9, 9E9, 9E9, 9E9]];
	VAR robtarget OpenholeUD_3969 := [[480.56, -5.1, 177.32], [0.059236, 0.704621, 0.691838, -0.14615], [0,0,0,0], [9E9, 9E9, 9E9, 9E9, 9E9, 9E9]];
	VAR robtarget OpenholeUD_3970 := [[484.52, -5.1, 176.78], [0.071906, 0.703441, 0.689311, -0.157639], [0,0,0,0], [9E9, 9E9, 9E9, 9E9, 9E9, 9E9]];
	VAR robtarget OpenholeUD_3971 := [[488.48, -5.1, 176.25], [0.084311, 0.702062, 0.686669, -0.168777], [0,0,0,0], [9E9, 9E9, 9E9, 9E9, 9E9, 9E9]];
	VAR robtarget OpenholeUD_3972 := [[492.45, -5.1, 175.72], [0.096425, 0.700501, 0.683931, -0.179552], [0,0,0,0], [9E9, 9E9, 9E9, 9E9, 9E9, 9E9]];
	VAR robtarget OpenholeUD_3973 := [[496.41, -5.1, 175.19], [0.108229, 0.698775, 0.681114, -0.189957], [0,0,0,0], [9E9, 9E9, 9E9, 9E9, 9E9, 9E9]];
	VAR robtarget OpenholeUD_3974 := [[500.38, -5.1, 174.66], [0.119709, 0.6969, 0.678237, -0.199988], [0,0,0,0], [9E9, 9E9, 9E9, 9E9, 9E9, 9E9]];
	VAR robtarget OpenholeUD_3975 := [[504.34, -5.1, 174.13], [0.130851, 0.694894, 0.675314, -0.209644], [0,0,0,0], [9E9, 9E9, 9E9, 9E9, 9E9, 9E9]];
	VAR robtarget OpenholeUD_3976 := [[509.32, -5.1, 173.46], [0.183051, 0.683002, 0.683002, -0.183051], [0,0,0,0], [9E9, 9E9, 9E9, 9E9, 9E9, 9E9]];
	VAR robtarget OpenholeUD_3977 := [[513.32, -5.1, 173.45], [0.183051, 0.683002, 0.683002, -0.183051], [0,0,0,0], [9E9, 9E9, 9E9, 9E9, 9E9, 9E9]];
	VAR robtarget OpenholeUD_3978 := [[517.32, -5.1, 173.43], [0.183051, 0.683002, 0.683002, -0.183051], [0,0,0,0], [9E9, 9E9, 9E9, 9E9, 9E9, 9E9]];
	VAR robtarget OpenholeUD_3979 := [[521.32, -5.1, 173.42], [0.183051, 0.683002, 0.683002, -0.183051], [0,0,0,0], [9E9, 9E9, 9E9, 9E9, 9E9, 9E9]];
	VAR robtarget OpenholeUD_3980 := [[529.32, -5.1, 173.4], [0.183051, 0.683002, 0.683002, -0.183051], [0,0,0,0], [9E9, 9E9, 9E9, 9E9, 9E9, 9E9]];
	VAR robtarget OpenholeUD_3981 := [[529.32, -5.1, 173.4], [0.183051, 0.683002, 0.683002, -0.183051], [0,0,0,0], [9E9, 9E9, 9E9, 9E9, 9E9, 9E9]];
	VAR robtarget OpenholeUD_3982 := [[529.32, -3.9, 172.7], [0.183051, 0.683002, 0.683002, -0.183051], [0,0,0,0], [9E9, 9E9, 9E9, 9E9, 9E9, 9E9]];
	VAR robtarget OpenholeUD_3983 := [[525.32, -3.9, 172.72], [0.183051, 0.683002, 0.683002, -0.183051], [0,0,0,0], [9E9, 9E9, 9E9, 9E9, 9E9, 9E9]];
	VAR robtarget OpenholeUD_3984 := [[521.32, -3.9, 172.73], [0.183051, 0.683002, 0.683002, -0.183051], [0,0,0,0], [9E9, 9E9, 9E9, 9E9, 9E9, 9E9]];
	VAR robtarget OpenholeUD_3985 := [[517.32, -3.9, 172.74], [0.183051, 0.683002, 0.683002, -0.183051], [0,0,0,0], [9E9, 9E9, 9E9, 9E9, 9E9, 9E9]];
	VAR robtarget OpenholeUD_3986 := [[509.32, -3.9, 172.77], [0.183051, 0.683002, 0.683002, -0.183051], [0,0,0,0], [9E9, 9E9, 9E9, 9E9, 9E9, 9E9]];
	VAR robtarget OpenholeUD_3987 := [[505.36, -3.9, 173.34], [0.130176, 0.695021, 0.673488, -0.21544], [0,0,0,0], [9E9, 9E9, 9E9, 9E9, 9E9, 9E9]];
	VAR robtarget OpenholeUD_3988 := [[501.4, -3.9, 173.92], [0.119076, 0.697009, 0.676446, -0.205962], [0,0,0,0], [9E9, 9E9, 9E9, 9E9, 9E9, 9E9]];
	VAR robtarget OpenholeUD_3989 := [[497.44, -3.9, 174.5], [0.107639, 0.698866, 0.679368, -0.196109], [0,0,0,0], [9E9, 9E9, 9E9, 9E9, 9E9, 9E9]];
	VAR robtarget OpenholeUD_3990 := [[493.49, -3.9, 175.07], [0.095877, 0.700577, 0.682238, -0.18588], [0,0,0,0], [9E9, 9E9, 9E9, 9E9, 9E9, 9E9]];
	VAR robtarget OpenholeUD_3991 := [[489.53, -3.9, 175.65], [0.083805, 0.702123, 0.685038, -0.175279], [0,0,0,0], [9E9, 9E9, 9E9, 9E9, 9E9, 9E9]];
	VAR robtarget OpenholeUD_3992 := [[485.57, -3.9, 176.23], [0.071442, 0.703488, 0.687751, -0.164311], [0,0,0,0], [9E9, 9E9, 9E9, 9E9, 9E9, 9E9]];
	VAR robtarget OpenholeUD_3993 := [[481.61, -3.9, 176.8], [0.058811, 0.704657, 0.690359, -0.152987], [0,0,0,0], [9E9, 9E9, 9E9, 9E9, 9E9, 9E9]];
	VAR robtarget OpenholeUD_3994 := [[477.65, -3.9, 177.38], [0.045939, 0.705613, 0.692841, -0.141319], [0,0,0,0], [9E9, 9E9, 9E9, 9E9, 9E9, 9E9]];
	VAR robtarget OpenholeUD_3995 := [[473.7, -3.9, 177.95], [0.032857, 0.706343, 0.69518, -0.129325], [0,0,0,0], [9E9, 9E9, 9E9, 9E9, 9E9, 9E9]];
	VAR robtarget OpenholeUD_3996 := [[469.74, -3.9, 178.53], [0.019599, 0.706835, 0.697355, -0.117029], [0,0,0,0], [9E9, 9E9, 9E9, 9E9, 9E9, 9E9]];
	VAR robtarget OpenholeUD_3997 := [[465.78, -3.9, 179.11], [0.006204, 0.70708, 0.699349, -0.104455], [0,0,0,0], [9E9, 9E9, 9E9, 9E9, 9E9, 9E9]];
	VAR robtarget OpenholeUD_3998 := [[461.82, -3.9, 179.68], [-0.007287, 0.707069, 0.701144, -0.091635], [0,0,0,0], [9E9, 9E9, 9E9, 9E9, 9E9, 9E9]];
	VAR robtarget OpenholeUD_3999 := [[457.86, -3.9, 180.26], [-0.020833, 0.7068, 0.702725, -0.078602], [0,0,0,0], [9E9, 9E9, 9E9, 9E9, 9E9, 9E9]];
	VAR robtarget OpenholeUD_4000 := [[453.9, -3.9, 180.84], [-0.034388, 0.70627, 0.704076, -0.065394], [0,0,0,0], [9E9, 9E9, 9E9, 9E9, 9E9, 9E9]];
	VAR robtarget OpenholeUD_4001 := [[449.95, -3.9, 181.41], [-0.047907, 0.705482, 0.705188, -0.052051], [0,0,0,0], [9E9, 9E9, 9E9, 9E9, 9E9, 9E9]];
	VAR robtarget OpenholeUD_4002 := [[445.99, -3.9, 181.99], [-0.061347, 0.704441, 0.706052, -0.038616], [0,0,0,0], [9E9, 9E9, 9E9, 9E9, 9E9, 9E9]];
	VAR robtarget OpenholeUD_4003 := [[442.03, -3.9, 182.57], [-0.074663, 0.703154, 0.70666, -0.025132], [0,0,0,0], [9E9, 9E9, 9E9, 9E9, 9E9, 9E9]];
	VAR robtarget OpenholeUD_4004 := [[438.07, -3.9, 183.14], [-0.087814, 0.701633, 0.707011, -0.011642], [0,0,0,0], [9E9, 9E9, 9E9, 9E9, 9E9, 9E9]];
	VAR robtarget OpenholeUD_4005 := [[434.11, -3.9, 183.72], [-0.10076, 0.699891, 0.707104, 0.001809], [0,0,0,0], [9E9, 9E9, 9E9, 9E9, 9E9, 9E9]];
	VAR robtarget OpenholeUD_4006 := [[430.16, -3.9, 184.3], [-0.113466, 0.697944, 0.706944, 0.015179], [0,0,0,0], [9E9, 9E9, 9E9, 9E9, 9E9, 9E9]];
	VAR robtarget OpenholeUD_4007 := [[426.2, -3.9, 184.87], [-0.1259, 0.695808, 0.706535, 0.028426], [0,0,0,0], [9E9, 9E9, 9E9, 9E9, 9E9, 9E9]];
	VAR robtarget OpenholeUD_4008 := [[422.24, -3.9, 185.45], [-0.138034, 0.693503, 0.705887, 0.041514], [0,0,0,0], [9E9, 9E9, 9E9, 9E9, 9E9, 9E9]];
	VAR robtarget OpenholeUD_4009 := [[418.28, -3.9, 186.03], [-0.149844, 0.691048, 0.705011, 0.054405], [0,0,0,0], [9E9, 9E9, 9E9, 9E9, 9E9, 9E9]];
	VAR robtarget OpenholeUD_4010 := [[414.32, -3.9, 186.6], [-0.161311, 0.688461, 0.703919, 0.06707], [0,0,0,0], [9E9, 9E9, 9E9, 9E9, 9E9, 9E9]];
	VAR robtarget OpenholeUD_4011 := [[410.36, -3.9, 187.18], [-0.17242, 0.685763, 0.702626, 0.079479], [0,0,0,0], [9E9, 9E9, 9E9, 9E9, 9E9, 9E9]];
	VAR robtarget OpenholeUD_4012 := [[406.41, -3.9, 187.76], [-0.18316, 0.682973, 0.701148, 0.091609], [0,0,0,0], [9E9, 9E9, 9E9, 9E9, 9E9, 9E9]];
	VAR robtarget OpenholeUD_4013 := [[402.45, -3.9, 188.33], [-0.193524, 0.680109, 0.6995, 0.103438], [0,0,0,0], [9E9, 9E9, 9E9, 9E9, 9E9, 9E9]];
	VAR robtarget OpenholeUD_4014 := [[398.49, -3.9, 188.91], [-0.203509, 0.677188, 0.6977, 0.114952], [0,0,0,0], [9E9, 9E9, 9E9, 9E9, 9E9, 9E9]];
	VAR robtarget OpenholeUD_4015 := [[394.53, -3.9, 189.49], [-0.213115, 0.674227, 0.695765, 0.126137], [0,0,0,0], [9E9, 9E9, 9E9, 9E9, 9E9, 9E9]];
	VAR robtarget OpenholeUD_4016 := [[389.37, -3.9, 190.24], [-0.225065, 0.670332, 0.693068, 0.140202], [0,0,0,0], [9E9, 9E9, 9E9, 9E9, 9E9, 9E9]];
	VAR robtarget OpenholeUD_4017 := [[385.37, -3.9, 190.25], [-0.183051, 0.683002, 0.683002, 0.183051], [0,0,0,0], [9E9, 9E9, 9E9, 9E9, 9E9, 9E9]];
	VAR robtarget OpenholeUD_4018 := [[381.37, -3.9, 190.26], [-0.183051, 0.683002, 0.683002, 0.183051], [0,0,0,0], [9E9, 9E9, 9E9, 9E9, 9E9, 9E9]];
	VAR robtarget OpenholeUD_4019 := [[377.37, -3.9, 190.27], [-0.183051, 0.683002, 0.683002, 0.183051], [0,0,0,0], [9E9, 9E9, 9E9, 9E9, 9E9, 9E9]];
	VAR robtarget OpenholeUD_4020 := [[373.37, -3.9, 190.29], [-0.183051, 0.683002, 0.683002, 0.183051], [0,0,0,0], [9E9, 9E9, 9E9, 9E9, 9E9, 9E9]];
	VAR robtarget OpenholeUD_4021 := [[369.37, -3.9, 190.3], [-0.183051, 0.683002, 0.683002, 0.183051], [0,0,0,0], [9E9, 9E9, 9E9, 9E9, 9E9, 9E9]];
	VAR robtarget OpenholeUD_4022 := [[369.37, -3.9, 190.3], [-0.183051, 0.683002, 0.683002, 0.183051], [0,0,0,0], [9E9, 9E9, 9E9, 9E9, 9E9, 9E9]];
	VAR robtarget OpenholeUD_4023 := [[369.38, -2.7, 190.99], [-0.183051, 0.683002, 0.683002, 0.183051], [0,0,0,0], [9E9, 9E9, 9E9, 9E9, 9E9, 9E9]];
	VAR robtarget OpenholeUD_4024 := [[373.38, -2.7, 190.98], [-0.183051, 0.683002, 0.683002, 0.183051], [0,0,0,0], [9E9, 9E9, 9E9, 9E9, 9E9, 9E9]];
	VAR robtarget OpenholeUD_4025 := [[377.38, -2.7, 190.97], [-0.183051, 0.683002, 0.683002, 0.183051], [0,0,0,0], [9E9, 9E9, 9E9, 9E9, 9E9, 9E9]];
	VAR robtarget OpenholeUD_4026 := [[381.38, -2.7, 190.96], [-0.183051, 0.683002, 0.683002, 0.183051], [0,0,0,0], [9E9, 9E9, 9E9, 9E9, 9E9, 9E9]];
	VAR robtarget OpenholeUD_4027 := [[385.38, -2.7, 190.94], [-0.183051, 0.683002, 0.683002, 0.183051], [0,0,0,0], [9E9, 9E9, 9E9, 9E9, 9E9, 9E9]];
	VAR robtarget OpenholeUD_4028 := [[389.38, -2.7, 190.93], [-0.228363, 0.669216, 0.693748, 0.136796], [0,0,0,0], [9E9, 9E9, 9E9, 9E9, 9E9, 9E9]];
	VAR robtarget OpenholeUD_4029 := [[393.33, -2.7, 190.31], [-0.219331, 0.672231, 0.695789, 0.126007], [0,0,0,0], [9E9, 9E9, 9E9, 9E9, 9E9, 9E9]];
	VAR robtarget OpenholeUD_4030 := [[397.28, -2.7, 189.69], [-0.209923, 0.675228, 0.697712, 0.114881], [0,0,0,0], [9E9, 9E9, 9E9, 9E9, 9E9, 9E9]];
	VAR robtarget OpenholeUD_4031 := [[401.23, -2.7, 189.07], [-0.200136, 0.678193, 0.699502, 0.103426], [0,0,0,0], [9E9, 9E9, 9E9, 9E9, 9E9, 9E9]];
	VAR robtarget OpenholeUD_4032 := [[405.18, -2.7, 188.44], [-0.18997, 0.681111, 0.701142, 0.091654], [0,0,0,0], [9E9, 9E9, 9E9, 9E9, 9E9, 9E9]];
	VAR robtarget OpenholeUD_4033 := [[409.13, -2.7, 187.82], [-0.179425, 0.683964, 0.702614, 0.079582], [0,0,0,0], [9E9, 9E9, 9E9, 9E9, 9E9, 9E9]];
	VAR robtarget OpenholeUD_4034 := [[413.08, -2.7, 187.2], [-0.168507, 0.686735, 0.703904, 0.067227], [0,0,0,0], [9E9, 9E9, 9E9, 9E9, 9E9, 9E9]];
	VAR robtarget OpenholeUD_4035 := [[417.04, -2.7, 186.58], [-0.157225, 0.689406, 0.704995, 0.054614], [0,0,0,0], [9E9, 9E9, 9E9, 9E9, 9E9, 9E9]];
	VAR robtarget OpenholeUD_4036 := [[420.99, -2.7, 185.96], [-0.145592, 0.691956, 0.705872, 0.04177], [0,0,0,0], [9E9, 9E9, 9E9, 9E9, 9E9, 9E9]];
	VAR robtarget OpenholeUD_4037 := [[424.94, -2.7, 185.34], [-0.133625, 0.694366, 0.706523, 0.028725], [0,0,0,0], [9E9, 9E9, 9E9, 9E9, 9E9, 9E9]];
	VAR robtarget OpenholeUD_4038 := [[428.89, -2.7, 184.72], [-0.121346, 0.696617, 0.706937, 0.015515], [0,0,0,0], [9E9, 9E9, 9E9, 9E9, 9E9, 9E9]];
	VAR robtarget OpenholeUD_4039 := [[432.84, -2.7, 184.1], [-0.108781, 0.698689, 0.707103, 0.002177], [0,0,0,0], [9E9, 9E9, 9E9, 9E9, 9E9, 9E9]];
	VAR robtarget OpenholeUD_4040 := [[436.79, -2.7, 183.48], [-0.09596, 0.700565, 0.707017, -0.01125], [0,0,0,0], [9E9, 9E9, 9E9, 9E9, 9E9, 9E9]];
	VAR robtarget OpenholeUD_4041 := [[440.75, -2.7, 182.85], [-0.082918, 0.702228, 0.706674, -0.024722], [0,0,0,0], [9E9, 9E9, 9E9, 9E9, 9E9, 9E9]];
	VAR robtarget OpenholeUD_4042 := [[444.7, -2.7, 182.23], [-0.069691, 0.703664, 0.706074, -0.038196], [0,0,0,0], [9E9, 9E9, 9E9, 9E9, 9E9, 9E9]];
	VAR robtarget OpenholeUD_4043 := [[448.65, -2.7, 181.61], [-0.05632, 0.70486, 0.705219, -0.051629], [0,0,0,0], [9E9, 9E9, 9E9, 9E9, 9E9, 9E9]];
	VAR robtarget OpenholeUD_4044 := [[452.6, -2.7, 180.99], [-0.042847, 0.705807, 0.704115, -0.064977], [0,0,0,0], [9E9, 9E9, 9E9, 9E9, 9E9, 9E9]];
	VAR robtarget OpenholeUD_4045 := [[456.55, -2.7, 180.37], [-0.029318, 0.706499, 0.70277, -0.078198], [0,0,0,0], [9E9, 9E9, 9E9, 9E9, 9E9, 9E9]];
	VAR robtarget OpenholeUD_4046 := [[460.5, -2.7, 179.75], [-0.015777, 0.706931, 0.701194, -0.09125], [0,0,0,0], [9E9, 9E9, 9E9, 9E9, 9E9, 9E9]];
	VAR robtarget OpenholeUD_4047 := [[464.45, -2.7, 179.13], [-0.002268, 0.707103, 0.699403, -0.104096], [0,0,0,0], [9E9, 9E9, 9E9, 9E9, 9E9, 9E9]];
	VAR robtarget OpenholeUD_4048 := [[468.41, -2.7, 178.51], [0.011166, 0.707019, 0.69741, -0.116701], [0,0,0,0], [9E9, 9E9, 9E9, 9E9, 9E9, 9E9]];
	VAR robtarget OpenholeUD_4049 := [[472.36, -2.7, 177.88], [0.024482, 0.706683, 0.695234, -0.129035], [0,0,0,0], [9E9, 9E9, 9E9, 9E9, 9E9, 9E9]];
	VAR robtarget OpenholeUD_4050 := [[476.31, -2.7, 177.26], [0.037641, 0.706104, 0.692892, -0.14107], [0,0,0,0], [9E9, 9E9, 9E9, 9E9, 9E9, 9E9]];
	VAR robtarget OpenholeUD_4051 := [[480.26, -2.7, 176.64], [0.050608, 0.705293, 0.690404, -0.152782], [0,0,0,0], [9E9, 9E9, 9E9, 9E9, 9E9, 9E9]];
	VAR robtarget OpenholeUD_4052 := [[484.21, -2.7, 176.02], [0.063349, 0.704263, 0.687789, -0.164154], [0,0,0,0], [9E9, 9E9, 9E9, 9E9, 9E9, 9E9]];
	VAR robtarget OpenholeUD_4053 := [[488.16, -2.7, 175.4], [0.075837, 0.703028, 0.685066, -0.175171], [0,0,0,0], [9E9, 9E9, 9E9, 9E9, 9E9, 9E9]];
	VAR robtarget OpenholeUD_4054 := [[492.11, -2.7, 174.78], [0.088045, 0.701604, 0.682254, -0.185822], [0,0,0,0], [9E9, 9E9, 9E9, 9E9, 9E9, 9E9]];
	VAR robtarget OpenholeUD_4055 := [[496.07, -2.7, 174.16], [0.099954, 0.700007, 0.67937, -0.196101], [0,0,0,0], [9E9, 9E9, 9E9, 9E9, 9E9, 9E9]];
	VAR robtarget OpenholeUD_4056 := [[500.02, -2.7, 173.54], [0.111546, 0.698253, 0.676433, -0.206005], [0,0,0,0], [9E9, 9E9, 9E9, 9E9, 9E9, 9E9]];
	VAR robtarget OpenholeUD_4057 := [[503.97, -2.7, 172.91], [0.122809, 0.696361, 0.673458, -0.215533], [0,0,0,0], [9E9, 9E9, 9E9, 9E9, 9E9, 9E9]];
	VAR robtarget OpenholeUD_4058 := [[509.32, -2.7, 172.07], [0.183051, 0.683002, 0.683002, -0.183051], [0,0,0,0], [9E9, 9E9, 9E9, 9E9, 9E9, 9E9]];
	VAR robtarget OpenholeUD_4059 := [[513.32, -2.7, 172.06], [0.183051, 0.683002, 0.683002, -0.183051], [0,0,0,0], [9E9, 9E9, 9E9, 9E9, 9E9, 9E9]];
	VAR robtarget OpenholeUD_4060 := [[517.32, -2.7, 172.05], [0.183051, 0.683002, 0.683002, -0.183051], [0,0,0,0], [9E9, 9E9, 9E9, 9E9, 9E9, 9E9]];
	VAR robtarget OpenholeUD_4061 := [[521.32, -2.7, 172.04], [0.183051, 0.683002, 0.683002, -0.183051], [0,0,0,0], [9E9, 9E9, 9E9, 9E9, 9E9, 9E9]];
	VAR robtarget OpenholeUD_4062 := [[525.32, -2.7, 172.02], [0.183051, 0.683002, 0.683002, -0.183051], [0,0,0,0], [9E9, 9E9, 9E9, 9E9, 9E9, 9E9]];
	VAR robtarget OpenholeUD_4063 := [[529.32, -2.7, 172.01], [0.183051, 0.683002, 0.683002, -0.183051], [0,0,0,0], [9E9, 9E9, 9E9, 9E9, 9E9, 9E9]];
	VAR robtarget OpenholeUD_4064 := [[529.32, -2.7, 172.01], [0.183051, 0.683002, 0.683002, -0.183051], [0,0,0,0], [9E9, 9E9, 9E9, 9E9, 9E9, 9E9]];
	VAR robtarget OpenholeUD_4065 := [[529.32, -1.5, 171.32], [0.183051, 0.683002, 0.683002, -0.183051], [0,0,0,0], [9E9, 9E9, 9E9, 9E9, 9E9, 9E9]];
	VAR robtarget OpenholeUD_4066 := [[525.32, -1.5, 171.33], [0.183051, 0.683002, 0.683002, -0.183051], [0,0,0,0], [9E9, 9E9, 9E9, 9E9, 9E9, 9E9]];
	VAR robtarget OpenholeUD_4067 := [[521.32, -1.5, 171.34], [0.183051, 0.683002, 0.683002, -0.183051], [0,0,0,0], [9E9, 9E9, 9E9, 9E9, 9E9, 9E9]];
	VAR robtarget OpenholeUD_4068 := [[517.32, -1.5, 171.35], [0.183051, 0.683002, 0.683002, -0.183051], [0,0,0,0], [9E9, 9E9, 9E9, 9E9, 9E9, 9E9]];
	VAR robtarget OpenholeUD_4069 := [[513.32, -1.5, 171.37], [0.183051, 0.683002, 0.683002, -0.183051], [0,0,0,0], [9E9, 9E9, 9E9, 9E9, 9E9, 9E9]];
	VAR robtarget OpenholeUD_4070 := [[509.32, -1.5, 171.38], [0.183051, 0.683002, 0.683002, -0.183051], [0,0,0,0], [9E9, 9E9, 9E9, 9E9, 9E9, 9E9]];
	VAR robtarget OpenholeUD_4071 := [[505.37, -1.5, 172.05], [0.123254, 0.696282, 0.671297, -0.222172], [0,0,0,0], [9E9, 9E9, 9E9, 9E9, 9E9, 9E9]];
	VAR robtarget OpenholeUD_4072 := [[501.43, -1.5, 172.71], [0.112069, 0.698169, 0.674308, -0.21286], [0,0,0,0], [9E9, 9E9, 9E9, 9E9, 9E9, 9E9]];
	VAR robtarget OpenholeUD_4073 := [[497.48, -1.5, 173.38], [0.100554, 0.699921, 0.677289, -0.203173], [0,0,0,0], [9E9, 9E9, 9E9, 9E9, 9E9, 9E9]];
	VAR robtarget OpenholeUD_4074 := [[493.54, -1.5, 174.04], [0.088722, 0.701519, 0.680227, -0.193109], [0,0,0,0], [9E9, 9E9, 9E9, 9E9, 9E9, 9E9]];
	VAR robtarget OpenholeUD_4075 := [[489.59, -1.5, 174.71], [0.076587, 0.702947, 0.683104, -0.182671], [0,0,0,0], [9E9, 9E9, 9E9, 9E9, 9E9, 9E9]];
	VAR robtarget OpenholeUD_4076 := [[485.65, -1.5, 175.37], [0.064169, 0.704189, 0.685903, -0.171862], [0,0,0,0], [9E9, 9E9, 9E9, 9E9, 9E9, 9E9]];
	VAR robtarget OpenholeUD_4077 := [[481.71, -1.5, 176.04], [0.051493, 0.705229, 0.688606, -0.160693], [0,0,0,0], [9E9, 9E9, 9E9, 9E9, 9E9, 9E9]];
	VAR robtarget OpenholeUD_4078 := [[477.76, -1.5, 176.71], [0.038587, 0.706053, 0.691192, -0.149174], [0,0,0,0], [9E9, 9E9, 9E9, 9E9, 9E9, 9E9]];
	VAR robtarget OpenholeUD_4079 := [[473.82, -1.5, 177.37], [0.025481, 0.706648, 0.693644, -0.137323], [0,0,0,0], [9E9, 9E9, 9E9, 9E9, 9E9, 9E9]];
	VAR robtarget OpenholeUD_4080 := [[469.87, -1.5, 178.04], [0.012211, 0.707001, 0.695942, -0.12516], [0,0,0,0], [9E9, 9E9, 9E9, 9E9, 9E9, 9E9]];
	VAR robtarget OpenholeUD_4081 := [[465.93, -1.5, 178.7], [-0.001185, 0.707106, 0.698066, -0.112711], [0,0,0,0], [9E9, 9E9, 9E9, 9E9, 9E9, 9E9]];
	VAR robtarget OpenholeUD_4082 := [[461.98, -1.5, 179.37], [-0.014665, 0.706955, 0.7, -0.100003], [0,0,0,0], [9E9, 9E9, 9E9, 9E9, 9E9, 9E9]];
	VAR robtarget OpenholeUD_4083 := [[458.04, -1.5, 180.03], [-0.028188, 0.706545, 0.701725, -0.087071], [0,0,0,0], [9E9, 9E9, 9E9, 9E9, 9E9, 9E9]];
	VAR robtarget OpenholeUD_4084 := [[454.1, -1.5, 180.7], [-0.041708, 0.705876, 0.703229, -0.073951], [0,0,0,0], [9E9, 9E9, 9E9, 9E9, 9E9, 9E9]];
	VAR robtarget OpenholeUD_4085 := [[450.15, -1.5, 181.37], [-0.055182, 0.70495, 0.704498, -0.060681], [0,0,0,0], [9E9, 9E9, 9E9, 9E9, 9E9, 9E9]];
	VAR robtarget OpenholeUD_4086 := [[446.21, -1.5, 182.03], [-0.068564, 0.703775, 0.705523, -0.047303], [0,0,0,0], [9E9, 9E9, 9E9, 9E9, 9E9, 9E9]];
	VAR robtarget OpenholeUD_4087 := [[442.26, -1.5, 182.7], [-0.081812, 0.702358, 0.706296, -0.03386], [0,0,0,0], [9E9, 9E9, 9E9, 9E9, 9E9, 9E9]];
	VAR robtarget OpenholeUD_4088 := [[438.32, -1.5, 183.36], [-0.094885, 0.700712, 0.706813, -0.020396], [0,0,0,0], [9E9, 9E9, 9E9, 9E9, 9E9, 9E9]];
	VAR robtarget OpenholeUD_4089 := [[434.38, -1.5, 184.03], [-0.107745, 0.69885, 0.707073, -0.006955], [0,0,0,0], [9E9, 9E9, 9E9, 9E9, 9E9, 9E9]];
	VAR robtarget OpenholeUD_4090 := [[430.43, -1.5, 184.69], [-0.120356, 0.696789, 0.707078, 0.006421], [0,0,0,0], [9E9, 9E9, 9E9, 9E9, 9E9, 9E9]];
	VAR robtarget OpenholeUD_4091 := [[426.49, -1.5, 185.36], [-0.132688, 0.694546, 0.706833, 0.019691], [0,0,0,0], [9E9, 9E9, 9E9, 9E9, 9E9, 9E9]];
	VAR robtarget OpenholeUD_4092 := [[422.54, -1.5, 186.03], [-0.144714, 0.69214, 0.706345, 0.032816], [0,0,0,0], [9E9, 9E9, 9E9, 9E9, 9E9, 9E9]];
	VAR robtarget OpenholeUD_4093 := [[418.6, -1.5, 186.69], [-0.15641, 0.689591, 0.705625, 0.045759], [0,0,0,0], [9E9, 9E9, 9E9, 9E9, 9E9, 9E9]];
	VAR robtarget OpenholeUD_4094 := [[414.65, -1.5, 187.36], [-0.167759, 0.686918, 0.704684, 0.058488], [0,0,0,0], [9E9, 9E9, 9E9, 9E9, 9E9, 9E9]];
	VAR robtarget OpenholeUD_4095 := [[410.71, -1.5, 188.02], [-0.178746, 0.684142, 0.703536, 0.070975], [0,0,0,0], [9E9, 9E9, 9E9, 9E9, 9E9, 9E9]];
	VAR robtarget OpenholeUD_4096 := [[406.77, -1.5, 188.69], [-0.189362, 0.68128, 0.702196, 0.083193], [0,0,0,0], [9E9, 9E9, 9E9, 9E9, 9E9, 9E9]];
	VAR robtarget OpenholeUD_4097 := [[402.82, -1.5, 189.35], [-0.1996, 0.678351, 0.70068, 0.095122], [0,0,0,0], [9E9, 9E9, 9E9, 9E9, 9E9, 9E9]];
	VAR robtarget OpenholeUD_4098 := [[398.88, -1.5, 190.02], [-0.209458, 0.675372, 0.699003, 0.106744], [0,0,0,0], [9E9, 9E9, 9E9, 9E9, 9E9, 9E9]];
	VAR robtarget OpenholeUD_4099 := [[394.93, -1.5, 190.69], [-0.218936, 0.672359, 0.697184, 0.118044], [0,0,0,0], [9E9, 9E9, 9E9, 9E9, 9E9, 9E9]];
	VAR robtarget OpenholeUD_4100 := [[389.38, -1.5, 191.62], [-0.231647, 0.668087, 0.69441, 0.133396], [0,0,0,0], [9E9, 9E9, 9E9, 9E9, 9E9, 9E9]];
	VAR robtarget OpenholeUD_4101 := [[385.38, -1.5, 191.64], [-0.183051, 0.683002, 0.683002, 0.183051], [0,0,0,0], [9E9, 9E9, 9E9, 9E9, 9E9, 9E9]];
	VAR robtarget OpenholeUD_4102 := [[381.38, -1.5, 191.65], [-0.183051, 0.683002, 0.683002, 0.183051], [0,0,0,0], [9E9, 9E9, 9E9, 9E9, 9E9, 9E9]];
	VAR robtarget OpenholeUD_4103 := [[377.38, -1.5, 191.66], [-0.183051, 0.683002, 0.683002, 0.183051], [0,0,0,0], [9E9, 9E9, 9E9, 9E9, 9E9, 9E9]];
	VAR robtarget OpenholeUD_4104 := [[373.38, -1.5, 191.67], [-0.183051, 0.683002, 0.683002, 0.183051], [0,0,0,0], [9E9, 9E9, 9E9, 9E9, 9E9, 9E9]];
	VAR robtarget OpenholeUD_4105 := [[369.38, -1.5, 191.69], [-0.183051, 0.683002, 0.683002, 0.183051], [0,0,0,0], [9E9, 9E9, 9E9, 9E9, 9E9, 9E9]];
	VAR robtarget OpenholeUD_4106 := [[369.38, -1.5, 191.69], [-0.183051, 0.683002, 0.683002, 0.183051], [0,0,0,0], [9E9, 9E9, 9E9, 9E9, 9E9, 9E9]];
	VAR robtarget OpenholeUD_4107 := [[369.38, -0.3, 192.38], [-0.183051, 0.683002, 0.683002, 0.183051], [0,0,0,0], [9E9, 9E9, 9E9, 9E9, 9E9, 9E9]];
